  PROC Part73()
    MoveL Offs(pOrigin,152.4,74.3,0.0),vDraw,z1,tPen\WObj:=wPaper;
    MoveL Offs(pOrigin,152.2,74.1,0.0),vDraw,z1,tPen\WObj:=wPaper;
    MoveL Offs(pOrigin,152.2,73.8,0.0),vDraw,z1,tPen\WObj:=wPaper;
    MoveL Offs(pOrigin,152.0,73.6,0.0),vDraw,z1,tPen\WObj:=wPaper;
    MoveL Offs(pOrigin,152.0,73.0,0.0),vDraw,z1,tPen\WObj:=wPaper;
    MoveL Offs(pOrigin,151.8,72.8,0.0),vDraw,z1,tPen\WObj:=wPaper;
    MoveL Offs(pOrigin,151.8,72.4,0.0),vDraw,z1,tPen\WObj:=wPaper;
    MoveL Offs(pOrigin,151.6,72.2,0.0),vDraw,z1,tPen\WObj:=wPaper;
    MoveL Offs(pOrigin,151.6,71.9,0.0),vDraw,z1,tPen\WObj:=wPaper;
    MoveL Offs(pOrigin,151.4,71.7,0.0),vDraw,z1,tPen\WObj:=wPaper;
    MoveL Offs(pOrigin,151.4,71.3,0.0),vDraw,z1,tPen\WObj:=wPaper;
    MoveL Offs(pOrigin,151.3,71.1,0.0),vDraw,z1,tPen\WObj:=wPaper;
    MoveL Offs(pOrigin,151.3,70.7,0.0),vDraw,z1,tPen\WObj:=wPaper;
    MoveL Offs(pOrigin,151.1,70.5,0.0),vDraw,z1,tPen\WObj:=wPaper;
    MoveL Offs(pOrigin,151.1,70.0,0.0),vDraw,z1,tPen\WObj:=wPaper;
    MoveL Offs(pOrigin,150.9,69.8,0.0),vDraw,z1,tPen\WObj:=wPaper;
    MoveL Offs(pOrigin,150.9,69.4,0.0),vDraw,z1,tPen\WObj:=wPaper;
    MoveL Offs(pOrigin,150.7,69.2,0.0),vDraw,z1,tPen\WObj:=wPaper;
    MoveL Offs(pOrigin,150.7,68.8,0.0),vDraw,z1,tPen\WObj:=wPaper;
    MoveL Offs(pOrigin,150.5,68.7,0.0),vDraw,z1,tPen\WObj:=wPaper;
    MoveL Offs(pOrigin,150.5,68.3,0.0),vDraw,z1,tPen\WObj:=wPaper;
    MoveL Offs(pOrigin,150.3,68.1,0.0),vDraw,z1,tPen\WObj:=wPaper;
    MoveL Offs(pOrigin,150.3,67.7,0.0),vDraw,z1,tPen\WObj:=wPaper;
    MoveL Offs(pOrigin,150.1,67.5,0.0),vDraw,z1,tPen\WObj:=wPaper;
    MoveL Offs(pOrigin,150.1,67.0,0.0),vDraw,z1,tPen\WObj:=wPaper;
    MoveL Offs(pOrigin,149.9,66.8,0.0),vDraw,z1,tPen\WObj:=wPaper;
    MoveL Offs(pOrigin,149.9,66.4,0.0),vDraw,z1,tPen\WObj:=wPaper;
    MoveL Offs(pOrigin,149.7,66.2,0.0),vDraw,z1,tPen\WObj:=wPaper;
    MoveL Offs(pOrigin,149.7,65.8,0.0),vDraw,z1,tPen\WObj:=wPaper;
    MoveL Offs(pOrigin,149.6,65.6,0.0),vDraw,z1,tPen\WObj:=wPaper;
    MoveL Offs(pOrigin,149.6,65.3,0.0),vDraw,z1,tPen\WObj:=wPaper;
    MoveL Offs(pOrigin,149.4,65.1,0.0),vDraw,z1,tPen\WObj:=wPaper;
    MoveL Offs(pOrigin,149.4,64.7,0.0),vDraw,z1,tPen\WObj:=wPaper;
    MoveL Offs(pOrigin,149.2,64.5,0.0),vDraw,z1,tPen\WObj:=wPaper;
    MoveL Offs(pOrigin,149.2,64.1,0.0),vDraw,z1,tPen\WObj:=wPaper;
    MoveL Offs(pOrigin,149.0,63.9,0.0),vDraw,z1,tPen\WObj:=wPaper;
    MoveL Offs(pOrigin,149.0,63.6,0.0),vDraw,z1,tPen\WObj:=wPaper;
    MoveL Offs(pOrigin,148.8,63.4,0.0),vDraw,z1,tPen\WObj:=wPaper;
    MoveL Offs(pOrigin,148.8,63.0,0.0),vDraw,z1,tPen\WObj:=wPaper;
    MoveL Offs(pOrigin,148.6,62.8,0.0),vDraw,z1,tPen\WObj:=wPaper;
    MoveL Offs(pOrigin,148.6,62.4,0.0),vDraw,z1,tPen\WObj:=wPaper;
    MoveL Offs(pOrigin,148.4,62.2,0.0),vDraw,z1,tPen\WObj:=wPaper;
    MoveL Offs(pOrigin,148.4,61.7,0.0),vDraw,z1,tPen\WObj:=wPaper;
    MoveL Offs(pOrigin,148.2,61.5,0.0),vDraw,z1,tPen\WObj:=wPaper;
    MoveL Offs(pOrigin,148.2,61.1,0.0),vDraw,z1,tPen\WObj:=wPaper;
    MoveL Offs(pOrigin,148.0,60.9,0.0),vDraw,z1,tPen\WObj:=wPaper;
    MoveL Offs(pOrigin,148.0,60.5,0.0),vDraw,z1,tPen\WObj:=wPaper;
    MoveL Offs(pOrigin,147.9,60.3,0.0),vDraw,z1,tPen\WObj:=wPaper;
    MoveL Offs(pOrigin,147.9,59.8,0.0),vDraw,z1,tPen\WObj:=wPaper;
    MoveL Offs(pOrigin,147.5,59.2,0.0),vDraw,z1,tPen\WObj:=wPaper;
    MoveL Offs(pOrigin,147.5,58.6,0.0),vDraw,z1,tPen\WObj:=wPaper;
    MoveL Offs(pOrigin,147.3,58.5,0.0),vDraw,z1,tPen\WObj:=wPaper;
    MoveL Offs(pOrigin,147.3,58.1,0.0),vDraw,z1,tPen\WObj:=wPaper;
    MoveL Offs(pOrigin,147.1,57.9,0.0),vDraw,z1,tPen\WObj:=wPaper;
    MoveL Offs(pOrigin,147.1,57.5,0.0),vDraw,z1,tPen\WObj:=wPaper;
    MoveL Offs(pOrigin,146.9,57.3,0.0),vDraw,z1,tPen\WObj:=wPaper;
    MoveL Offs(pOrigin,146.9,56.9,0.0),vDraw,z1,tPen\WObj:=wPaper;
    MoveL Offs(pOrigin,146.7,56.8,0.0),vDraw,z1,tPen\WObj:=wPaper;
    MoveL Offs(pOrigin,146.7,56.2,0.0),vDraw,z1,tPen\WObj:=wPaper;
    MoveL Offs(pOrigin,146.5,56.0,0.0),vDraw,z1,tPen\WObj:=wPaper;
    MoveL Offs(pOrigin,146.5,55.6,0.0),vDraw,z1,tPen\WObj:=wPaper;
    MoveL Offs(pOrigin,146.3,55.4,0.0),vDraw,z1,tPen\WObj:=wPaper;
    MoveL Offs(pOrigin,146.3,55.1,0.0),vDraw,z1,tPen\WObj:=wPaper;
    MoveL Offs(pOrigin,146.2,54.9,0.0),vDraw,z1,tPen\WObj:=wPaper;
    MoveL Offs(pOrigin,146.2,54.3,0.0),vDraw,z1,tPen\WObj:=wPaper;
    MoveL Offs(pOrigin,146.0,54.1,0.0),vDraw,z1,tPen\WObj:=wPaper;
    MoveL Offs(pOrigin,146.0,53.7,0.0),vDraw,z1,tPen\WObj:=wPaper;
    MoveL Offs(pOrigin,145.8,53.5,0.0),vDraw,z1,tPen\WObj:=wPaper;
    MoveL Offs(pOrigin,145.8,53.0,0.0),vDraw,z1,tPen\WObj:=wPaper;
    MoveL Offs(pOrigin,145.6,52.8,0.0),vDraw,z1,tPen\WObj:=wPaper;
    MoveL Offs(pOrigin,145.6,52.2,0.0),vDraw,z1,tPen\WObj:=wPaper;
    MoveL Offs(pOrigin,145.4,52.0,0.0),vDraw,z1,tPen\WObj:=wPaper;
    MoveL Offs(pOrigin,145.4,51.5,0.0),vDraw,z1,tPen\WObj:=wPaper;
    MoveL Offs(pOrigin,145.2,51.3,0.0),vDraw,z1,tPen\WObj:=wPaper;
    MoveL Offs(pOrigin,145.2,50.9,0.0),vDraw,z1,tPen\WObj:=wPaper;
    MoveL Offs(pOrigin,145.0,50.7,0.0),vDraw,z1,tPen\WObj:=wPaper;
    MoveL Offs(pOrigin,145.0,50.1,0.0),vDraw,z1,tPen\WObj:=wPaper;
    MoveL Offs(pOrigin,144.8,50.0,0.0),vDraw,z1,tPen\WObj:=wPaper;
    MoveL Offs(pOrigin,144.8,49.4,0.0),vDraw,z1,tPen\WObj:=wPaper;
    MoveL Offs(pOrigin,144.6,49.2,0.0),vDraw,z1,tPen\WObj:=wPaper;
    MoveL Offs(pOrigin,144.6,48.6,0.0),vDraw,z1,tPen\WObj:=wPaper;
    MoveL Offs(pOrigin,144.5,48.4,0.0),vDraw,z1,tPen\WObj:=wPaper;
    MoveL Offs(pOrigin,144.5,47.7,0.0),vDraw,z1,tPen\WObj:=wPaper;
    MoveL Offs(pOrigin,144.3,47.5,0.0),vDraw,z1,tPen\WObj:=wPaper;
    MoveL Offs(pOrigin,144.3,46.9,0.0),vDraw,z1,tPen\WObj:=wPaper;
    MoveL Offs(pOrigin,144.1,46.7,0.0),vDraw,z1,tPen\WObj:=wPaper;
    MoveL Offs(pOrigin,144.1,46.2,0.0),vDraw,z1,tPen\WObj:=wPaper;
    MoveL Offs(pOrigin,143.9,46.0,0.0),vDraw,z1,tPen\WObj:=wPaper;
    MoveL Offs(pOrigin,143.9,45.2,0.0),vDraw,z1,tPen\WObj:=wPaper;
    MoveL Offs(pOrigin,143.7,45.0,0.0),vDraw,z1,tPen\WObj:=wPaper;
    MoveL Offs(pOrigin,143.7,44.3,0.0),vDraw,z1,tPen\WObj:=wPaper;
    MoveL Offs(pOrigin,143.5,44.1,0.0),vDraw,z1,tPen\WObj:=wPaper;
    MoveL Offs(pOrigin,143.5,43.3,0.0),vDraw,z1,tPen\WObj:=wPaper;
    MoveL Offs(pOrigin,143.3,43.2,0.0),vDraw,z1,tPen\WObj:=wPaper;
    MoveL Offs(pOrigin,143.3,42.4,0.0),vDraw,z1,tPen\WObj:=wPaper;
    MoveL Offs(pOrigin,143.1,42.2,0.0),vDraw,z1,tPen\WObj:=wPaper;
    MoveL Offs(pOrigin,143.1,41.3,0.0),vDraw,z1,tPen\WObj:=wPaper;
    MoveL Offs(pOrigin,142.9,41.1,0.0),vDraw,z1,tPen\WObj:=wPaper;
    MoveL Offs(pOrigin,142.9,40.1,0.0),vDraw,z1,tPen\WObj:=wPaper;
    MoveL Offs(pOrigin,142.8,39.9,0.0),vDraw,z1,tPen\WObj:=wPaper;
    MoveL Offs(pOrigin,142.8,39.0,0.0),vDraw,z1,tPen\WObj:=wPaper;
    MoveL Offs(pOrigin,142.6,38.8,0.0),vDraw,z1,tPen\WObj:=wPaper;
    MoveL Offs(pOrigin,142.6,37.5,0.0),vDraw,z1,tPen\WObj:=wPaper;
    MoveL Offs(pOrigin,142.0,36.7,0.0),vDraw,z1,tPen\WObj:=wPaper;
    MoveL Offs(pOrigin,140.3,36.7,0.0),vDraw,z1,tPen\WObj:=wPaper;
    MoveL Offs(pOrigin,140.1,36.5,0.0),vDraw,z1,tPen\WObj:=wPaper;
    MoveL Offs(pOrigin,139.2,36.4,0.0),vDraw,z1,tPen\WObj:=wPaper;
    MoveL Offs(pOrigin,138.2,35.8,0.0),vDraw,fine,tPen\WObj:=wPaper;
    MoveL Offs(pOrigin,138.2,35.8,15.0),vApproach,z5,tPen\WObj:=wPaper;
    MoveL Offs(pOrigin,143.1,36.7,15.0),vTravel,z5,tPen\WObj:=wPaper;
    MoveL Offs(pOrigin,143.1,36.7,0.0),vApproach,fine,tPen\WObj:=wPaper;
    MoveL Offs(pOrigin,143.1,37.3,0.0),vDraw,z1,tPen\WObj:=wPaper;
    MoveL Offs(pOrigin,143.3,37.5,0.0),vDraw,z1,tPen\WObj:=wPaper;
    MoveL Offs(pOrigin,143.3,38.8,0.0),vDraw,z1,tPen\WObj:=wPaper;
    MoveL Offs(pOrigin,143.5,39.0,0.0),vDraw,z1,tPen\WObj:=wPaper;
    MoveL Offs(pOrigin,143.5,40.1,0.0),vDraw,z1,tPen\WObj:=wPaper;
    MoveL Offs(pOrigin,143.7,40.3,0.0),vDraw,z1,tPen\WObj:=wPaper;
    MoveL Offs(pOrigin,143.7,41.1,0.0),vDraw,z1,tPen\WObj:=wPaper;
    MoveL Offs(pOrigin,143.9,41.3,0.0),vDraw,z1,tPen\WObj:=wPaper;
    MoveL Offs(pOrigin,143.9,42.2,0.0),vDraw,z1,tPen\WObj:=wPaper;
  ENDPROC

  PROC Part74()
    MoveL Offs(pOrigin,144.1,42.4,0.0),vDraw,z1,tPen\WObj:=wPaper;
    MoveL Offs(pOrigin,144.1,43.2,0.0),vDraw,z1,tPen\WObj:=wPaper;
    MoveL Offs(pOrigin,144.3,43.3,0.0),vDraw,z1,tPen\WObj:=wPaper;
    MoveL Offs(pOrigin,144.3,44.1,0.0),vDraw,z1,tPen\WObj:=wPaper;
    MoveL Offs(pOrigin,144.5,44.3,0.0),vDraw,z1,tPen\WObj:=wPaper;
    MoveL Offs(pOrigin,144.5,45.0,0.0),vDraw,z1,tPen\WObj:=wPaper;
    MoveL Offs(pOrigin,144.6,45.2,0.0),vDraw,z1,tPen\WObj:=wPaper;
    MoveL Offs(pOrigin,144.6,45.8,0.0),vDraw,z1,tPen\WObj:=wPaper;
    MoveL Offs(pOrigin,144.8,46.0,0.0),vDraw,z1,tPen\WObj:=wPaper;
    MoveL Offs(pOrigin,144.8,46.6,0.0),vDraw,z1,tPen\WObj:=wPaper;
    MoveL Offs(pOrigin,145.0,46.7,0.0),vDraw,z1,tPen\WObj:=wPaper;
    MoveL Offs(pOrigin,145.0,47.5,0.0),vDraw,z1,tPen\WObj:=wPaper;
    MoveL Offs(pOrigin,145.2,47.7,0.0),vDraw,z1,tPen\WObj:=wPaper;
    MoveL Offs(pOrigin,145.2,48.3,0.0),vDraw,z1,tPen\WObj:=wPaper;
    MoveL Offs(pOrigin,145.4,48.4,0.0),vDraw,z1,tPen\WObj:=wPaper;
    MoveL Offs(pOrigin,145.4,49.0,0.0),vDraw,z1,tPen\WObj:=wPaper;
    MoveL Offs(pOrigin,145.8,49.6,0.0),vDraw,z1,tPen\WObj:=wPaper;
    MoveL Offs(pOrigin,146.0,49.4,0.0),vDraw,z1,tPen\WObj:=wPaper;
    MoveL Offs(pOrigin,146.0,47.9,0.0),vDraw,z1,tPen\WObj:=wPaper;
    MoveL Offs(pOrigin,145.8,47.7,0.0),vDraw,z1,tPen\WObj:=wPaper;
    MoveL Offs(pOrigin,145.8,42.8,0.0),vDraw,z1,tPen\WObj:=wPaper;
    MoveL Offs(pOrigin,146.0,42.6,0.0),vDraw,z1,tPen\WObj:=wPaper;
    MoveL Offs(pOrigin,146.0,40.5,0.0),vDraw,z1,tPen\WObj:=wPaper;
    MoveL Offs(pOrigin,146.2,40.3,0.0),vDraw,z1,tPen\WObj:=wPaper;
    MoveL Offs(pOrigin,146.2,39.2,0.0),vDraw,z1,tPen\WObj:=wPaper;
    MoveL Offs(pOrigin,146.3,39.0,0.0),vDraw,z1,tPen\WObj:=wPaper;
    MoveL Offs(pOrigin,146.3,38.2,0.0),vDraw,z1,tPen\WObj:=wPaper;
    MoveL Offs(pOrigin,146.5,38.1,0.0),vDraw,z1,tPen\WObj:=wPaper;
    MoveL Offs(pOrigin,146.5,37.5,0.0),vDraw,z1,tPen\WObj:=wPaper;
    MoveL Offs(pOrigin,146.7,37.3,0.0),vDraw,z1,tPen\WObj:=wPaper;
    MoveL Offs(pOrigin,146.7,36.7,0.0),vDraw,z1,tPen\WObj:=wPaper;
    MoveL Offs(pOrigin,146.7,38.1,0.0),vDraw,z1,tPen\WObj:=wPaper;
    MoveL Offs(pOrigin,146.5,38.2,0.0),vDraw,z1,tPen\WObj:=wPaper;
    MoveL Offs(pOrigin,146.5,39.4,0.0),vDraw,z1,tPen\WObj:=wPaper;
    MoveL Offs(pOrigin,146.3,39.6,0.0),vDraw,z1,tPen\WObj:=wPaper;
    MoveL Offs(pOrigin,146.3,41.1,0.0),vDraw,z1,tPen\WObj:=wPaper;
    MoveL Offs(pOrigin,146.2,41.3,0.0),vDraw,z1,tPen\WObj:=wPaper;
    MoveL Offs(pOrigin,146.2,50.9,0.0),vDraw,z1,tPen\WObj:=wPaper;
    MoveL Offs(pOrigin,146.3,51.1,0.0),vDraw,z1,tPen\WObj:=wPaper;
    MoveL Offs(pOrigin,146.3,52.2,0.0),vDraw,z1,tPen\WObj:=wPaper;
    MoveL Offs(pOrigin,146.5,52.4,0.0),vDraw,z1,tPen\WObj:=wPaper;
    MoveL Offs(pOrigin,146.5,53.4,0.0),vDraw,z1,tPen\WObj:=wPaper;
    MoveL Offs(pOrigin,146.7,53.5,0.0),vDraw,z1,tPen\WObj:=wPaper;
    MoveL Offs(pOrigin,146.7,54.1,0.0),vDraw,z1,tPen\WObj:=wPaper;
    MoveL Offs(pOrigin,146.9,54.3,0.0),vDraw,z1,tPen\WObj:=wPaper;
    MoveL Offs(pOrigin,146.9,54.7,0.0),vDraw,z1,tPen\WObj:=wPaper;
    MoveL Offs(pOrigin,147.3,55.1,0.0),vDraw,z1,tPen\WObj:=wPaper;
    MoveL Offs(pOrigin,147.9,55.1,0.0),vDraw,z1,tPen\WObj:=wPaper;
    MoveL Offs(pOrigin,148.0,55.2,0.0),vDraw,z1,tPen\WObj:=wPaper;
    MoveL Offs(pOrigin,148.8,55.2,0.0),vDraw,z1,tPen\WObj:=wPaper;
    MoveL Offs(pOrigin,149.0,55.4,0.0),vDraw,z1,tPen\WObj:=wPaper;
    MoveL Offs(pOrigin,149.7,55.4,0.0),vDraw,z1,tPen\WObj:=wPaper;
    MoveL Offs(pOrigin,149.9,55.6,0.0),vDraw,z1,tPen\WObj:=wPaper;
    MoveL Offs(pOrigin,150.5,55.6,0.0),vDraw,z1,tPen\WObj:=wPaper;
    MoveL Offs(pOrigin,150.7,55.8,0.0),vDraw,z1,tPen\WObj:=wPaper;
    MoveL Offs(pOrigin,151.4,55.8,0.0),vDraw,z1,tPen\WObj:=wPaper;
    MoveL Offs(pOrigin,151.6,56.0,0.0),vDraw,z1,tPen\WObj:=wPaper;
    MoveL Offs(pOrigin,152.2,56.0,0.0),vDraw,z1,tPen\WObj:=wPaper;
    MoveL Offs(pOrigin,152.4,56.2,0.0),vDraw,z1,tPen\WObj:=wPaper;
    MoveL Offs(pOrigin,153.0,56.2,0.0),vDraw,z1,tPen\WObj:=wPaper;
    MoveL Offs(pOrigin,153.1,56.4,0.0),vDraw,z1,tPen\WObj:=wPaper;
    MoveL Offs(pOrigin,153.7,56.4,0.0),vDraw,z1,tPen\WObj:=wPaper;
    MoveL Offs(pOrigin,153.9,56.6,0.0),vDraw,z1,tPen\WObj:=wPaper;
    MoveL Offs(pOrigin,154.5,56.6,0.0),vDraw,z1,tPen\WObj:=wPaper;
    MoveL Offs(pOrigin,154.7,56.8,0.0),vDraw,z1,tPen\WObj:=wPaper;
    MoveL Offs(pOrigin,155.4,56.8,0.0),vDraw,z1,tPen\WObj:=wPaper;
    MoveL Offs(pOrigin,155.6,56.9,0.0),vDraw,z1,tPen\WObj:=wPaper;
    MoveL Offs(pOrigin,156.0,56.9,0.0),vDraw,z1,tPen\WObj:=wPaper;
    MoveL Offs(pOrigin,156.2,57.1,0.0),vDraw,z1,tPen\WObj:=wPaper;
    MoveL Offs(pOrigin,156.9,57.1,0.0),vDraw,z1,tPen\WObj:=wPaper;
    MoveL Offs(pOrigin,157.1,57.3,0.0),vDraw,z1,tPen\WObj:=wPaper;
    MoveL Offs(pOrigin,157.5,57.3,0.0),vDraw,z1,tPen\WObj:=wPaper;
    MoveL Offs(pOrigin,157.7,57.5,0.0),vDraw,z1,tPen\WObj:=wPaper;
    MoveL Offs(pOrigin,158.2,57.5,0.0),vDraw,z1,tPen\WObj:=wPaper;
    MoveL Offs(pOrigin,158.4,57.7,0.0),vDraw,z1,tPen\WObj:=wPaper;
    MoveL Offs(pOrigin,159.0,57.7,0.0),vDraw,z1,tPen\WObj:=wPaper;
    MoveL Offs(pOrigin,159.2,57.9,0.0),vDraw,z1,tPen\WObj:=wPaper;
    MoveL Offs(pOrigin,159.8,57.9,0.0),vDraw,z1,tPen\WObj:=wPaper;
    MoveL Offs(pOrigin,159.9,58.1,0.0),vDraw,z1,tPen\WObj:=wPaper;
    MoveL Offs(pOrigin,160.5,58.1,0.0),vDraw,z1,tPen\WObj:=wPaper;
    MoveL Offs(pOrigin,160.7,58.3,0.0),vDraw,z1,tPen\WObj:=wPaper;
    MoveL Offs(pOrigin,161.3,58.3,0.0),vDraw,z1,tPen\WObj:=wPaper;
    MoveL Offs(pOrigin,161.5,58.5,0.0),vDraw,z1,tPen\WObj:=wPaper;
    MoveL Offs(pOrigin,161.8,58.5,0.0),vDraw,z1,tPen\WObj:=wPaper;
    MoveL Offs(pOrigin,162.0,58.6,0.0),vDraw,z1,tPen\WObj:=wPaper;
    MoveL Offs(pOrigin,162.6,58.6,0.0),vDraw,z1,tPen\WObj:=wPaper;
    MoveL Offs(pOrigin,162.8,58.8,0.0),vDraw,z1,tPen\WObj:=wPaper;
    MoveL Offs(pOrigin,163.3,58.8,0.0),vDraw,z1,tPen\WObj:=wPaper;
    MoveL Offs(pOrigin,163.5,59.0,0.0),vDraw,z1,tPen\WObj:=wPaper;
    MoveL Offs(pOrigin,164.1,59.0,0.0),vDraw,z1,tPen\WObj:=wPaper;
    MoveL Offs(pOrigin,164.3,59.2,0.0),vDraw,z1,tPen\WObj:=wPaper;
    MoveL Offs(pOrigin,164.7,59.2,0.0),vDraw,z1,tPen\WObj:=wPaper;
    MoveL Offs(pOrigin,164.9,59.4,0.0),vDraw,z1,tPen\WObj:=wPaper;
    MoveL Offs(pOrigin,165.2,59.4,0.0),vDraw,z1,tPen\WObj:=wPaper;
    MoveL Offs(pOrigin,165.4,59.6,0.0),vDraw,z1,tPen\WObj:=wPaper;
    MoveL Offs(pOrigin,166.0,59.6,0.0),vDraw,z1,tPen\WObj:=wPaper;
    MoveL Offs(pOrigin,166.2,59.8,0.0),vDraw,z1,tPen\WObj:=wPaper;
    MoveL Offs(pOrigin,166.6,59.8,0.0),vDraw,z1,tPen\WObj:=wPaper;
    MoveL Offs(pOrigin,166.7,60.0,0.0),vDraw,z1,tPen\WObj:=wPaper;
    MoveL Offs(pOrigin,167.3,60.0,0.0),vDraw,z1,tPen\WObj:=wPaper;
    MoveL Offs(pOrigin,167.5,60.2,0.0),vDraw,z1,tPen\WObj:=wPaper;
    MoveL Offs(pOrigin,168.1,60.2,0.0),vDraw,z1,tPen\WObj:=wPaper;
    MoveL Offs(pOrigin,168.3,60.3,0.0),vDraw,z1,tPen\WObj:=wPaper;
    MoveL Offs(pOrigin,168.6,60.3,0.0),vDraw,z1,tPen\WObj:=wPaper;
    MoveL Offs(pOrigin,168.8,60.5,0.0),vDraw,z1,tPen\WObj:=wPaper;
    MoveL Offs(pOrigin,169.2,60.5,0.0),vDraw,z1,tPen\WObj:=wPaper;
    MoveL Offs(pOrigin,169.4,60.7,0.0),vDraw,z1,tPen\WObj:=wPaper;
    MoveL Offs(pOrigin,169.8,60.7,0.0),vDraw,z1,tPen\WObj:=wPaper;
    MoveL Offs(pOrigin,170.0,60.9,0.0),vDraw,z1,tPen\WObj:=wPaper;
    MoveL Offs(pOrigin,170.5,60.9,0.0),vDraw,z1,tPen\WObj:=wPaper;
    MoveL Offs(pOrigin,171.1,61.3,0.0),vDraw,z1,tPen\WObj:=wPaper;
    MoveL Offs(pOrigin,172.0,61.5,0.0),vDraw,z1,tPen\WObj:=wPaper;
    MoveL Offs(pOrigin,172.2,61.7,0.0),vDraw,z1,tPen\WObj:=wPaper;
    MoveL Offs(pOrigin,172.4,61.7,0.0),vDraw,z1,tPen\WObj:=wPaper;
    MoveL Offs(pOrigin,172.8,62.2,0.0),vDraw,z1,tPen\WObj:=wPaper;
    MoveL Offs(pOrigin,172.8,66.8,0.0),vDraw,z1,tPen\WObj:=wPaper;
    MoveL Offs(pOrigin,172.6,67.0,0.0),vDraw,z1,tPen\WObj:=wPaper;
    MoveL Offs(pOrigin,172.6,67.5,0.0),vDraw,z1,tPen\WObj:=wPaper;
    MoveL Offs(pOrigin,172.4,67.7,0.0),vDraw,z1,tPen\WObj:=wPaper;
    MoveL Offs(pOrigin,171.8,67.7,0.0),vDraw,z1,tPen\WObj:=wPaper;
  ENDPROC

  PROC Part75()
    MoveL Offs(pOrigin,171.7,67.5,0.0),vDraw,z1,tPen\WObj:=wPaper;
    MoveL Offs(pOrigin,171.3,67.5,0.0),vDraw,z1,tPen\WObj:=wPaper;
    MoveL Offs(pOrigin,171.1,67.3,0.0),vDraw,z1,tPen\WObj:=wPaper;
    MoveL Offs(pOrigin,170.7,67.3,0.0),vDraw,z1,tPen\WObj:=wPaper;
    MoveL Offs(pOrigin,170.5,67.1,0.0),vDraw,z1,tPen\WObj:=wPaper;
    MoveL Offs(pOrigin,170.0,67.1,0.0),vDraw,z1,tPen\WObj:=wPaper;
    MoveL Offs(pOrigin,169.8,67.0,0.0),vDraw,z1,tPen\WObj:=wPaper;
    MoveL Offs(pOrigin,169.4,67.0,0.0),vDraw,z1,tPen\WObj:=wPaper;
    MoveL Offs(pOrigin,169.2,66.8,0.0),vDraw,z1,tPen\WObj:=wPaper;
    MoveL Offs(pOrigin,168.8,66.8,0.0),vDraw,z1,tPen\WObj:=wPaper;
    MoveL Offs(pOrigin,168.6,66.6,0.0),vDraw,z1,tPen\WObj:=wPaper;
    MoveL Offs(pOrigin,168.1,66.6,0.0),vDraw,z1,tPen\WObj:=wPaper;
    MoveL Offs(pOrigin,167.9,66.4,0.0),vDraw,z1,tPen\WObj:=wPaper;
    MoveL Offs(pOrigin,167.7,66.4,0.0),vDraw,z1,tPen\WObj:=wPaper;
    MoveL Offs(pOrigin,167.5,66.6,0.0),vDraw,z1,tPen\WObj:=wPaper;
    MoveL Offs(pOrigin,168.8,67.9,0.0),vDraw,z1,tPen\WObj:=wPaper;
    MoveL Offs(pOrigin,169.0,67.9,0.0),vDraw,z1,tPen\WObj:=wPaper;
    MoveL Offs(pOrigin,169.8,68.7,0.0),vDraw,z1,tPen\WObj:=wPaper;
    MoveL Offs(pOrigin,170.0,68.7,0.0),vDraw,z1,tPen\WObj:=wPaper;
    MoveL Offs(pOrigin,170.7,69.4,0.0),vDraw,z1,tPen\WObj:=wPaper;
    MoveL Offs(pOrigin,170.9,69.4,0.0),vDraw,z1,tPen\WObj:=wPaper;
    MoveL Offs(pOrigin,171.5,70.0,0.0),vDraw,z1,tPen\WObj:=wPaper;
    MoveL Offs(pOrigin,171.7,70.0,0.0),vDraw,z1,tPen\WObj:=wPaper;
    MoveL Offs(pOrigin,172.4,70.7,0.0),vDraw,z1,tPen\WObj:=wPaper;
    MoveL Offs(pOrigin,172.6,70.7,0.0),vDraw,z1,tPen\WObj:=wPaper;
    MoveL Offs(pOrigin,173.0,71.1,0.0),vDraw,z1,tPen\WObj:=wPaper;
    MoveL Offs(pOrigin,172.8,70.9,0.0),vDraw,z1,tPen\WObj:=wPaper;
    MoveL Offs(pOrigin,171.8,70.5,0.0),vDraw,z1,tPen\WObj:=wPaper;
    MoveL Offs(pOrigin,171.5,70.2,0.0),vDraw,z1,tPen\WObj:=wPaper;
    MoveL Offs(pOrigin,171.3,70.2,0.0),vDraw,z1,tPen\WObj:=wPaper;
    MoveL Offs(pOrigin,170.9,69.8,0.0),vDraw,z1,tPen\WObj:=wPaper;
    MoveL Offs(pOrigin,170.7,69.8,0.0),vDraw,z1,tPen\WObj:=wPaper;
    MoveL Offs(pOrigin,170.3,69.4,0.0),vDraw,z1,tPen\WObj:=wPaper;
    MoveL Offs(pOrigin,170.1,69.4,0.0),vDraw,z1,tPen\WObj:=wPaper;
    MoveL Offs(pOrigin,168.3,67.7,0.0),vDraw,z1,tPen\WObj:=wPaper;
    MoveL Offs(pOrigin,168.1,67.7,0.0),vDraw,z1,tPen\WObj:=wPaper;
    MoveL Offs(pOrigin,166.4,66.0,0.0),vDraw,z1,tPen\WObj:=wPaper;
    MoveL Offs(pOrigin,166.2,66.0,0.0),vDraw,z1,tPen\WObj:=wPaper;
    MoveL Offs(pOrigin,166.0,65.8,0.0),vDraw,z1,tPen\WObj:=wPaper;
    MoveL Offs(pOrigin,165.4,65.8,0.0),vDraw,z1,tPen\WObj:=wPaper;
    MoveL Offs(pOrigin,165.2,65.6,0.0),vDraw,z1,tPen\WObj:=wPaper;
    MoveL Offs(pOrigin,164.9,65.6,0.0),vDraw,z1,tPen\WObj:=wPaper;
    MoveL Offs(pOrigin,164.7,65.4,0.0),vDraw,z1,tPen\WObj:=wPaper;
    MoveL Offs(pOrigin,164.1,65.4,0.0),vDraw,z1,tPen\WObj:=wPaper;
    MoveL Offs(pOrigin,163.9,65.3,0.0),vDraw,z1,tPen\WObj:=wPaper;
    MoveL Offs(pOrigin,163.5,65.3,0.0),vDraw,z1,tPen\WObj:=wPaper;
    MoveL Offs(pOrigin,163.3,65.1,0.0),vDraw,z1,tPen\WObj:=wPaper;
    MoveL Offs(pOrigin,162.8,65.1,0.0),vDraw,z1,tPen\WObj:=wPaper;
    MoveL Offs(pOrigin,162.6,64.9,0.0),vDraw,z1,tPen\WObj:=wPaper;
    MoveL Offs(pOrigin,162.0,64.9,0.0),vDraw,z1,tPen\WObj:=wPaper;
    MoveL Offs(pOrigin,161.8,64.7,0.0),vDraw,z1,tPen\WObj:=wPaper;
    MoveL Offs(pOrigin,161.5,64.7,0.0),vDraw,z1,tPen\WObj:=wPaper;
    MoveL Offs(pOrigin,161.3,64.5,0.0),vDraw,z1,tPen\WObj:=wPaper;
    MoveL Offs(pOrigin,160.9,64.5,0.0),vDraw,z1,tPen\WObj:=wPaper;
    MoveL Offs(pOrigin,160.7,64.3,0.0),vDraw,z1,tPen\WObj:=wPaper;
    MoveL Offs(pOrigin,160.1,64.3,0.0),vDraw,z1,tPen\WObj:=wPaper;
    MoveL Offs(pOrigin,159.9,64.1,0.0),vDraw,z1,tPen\WObj:=wPaper;
    MoveL Offs(pOrigin,159.4,64.1,0.0),vDraw,z1,tPen\WObj:=wPaper;
    MoveL Offs(pOrigin,159.2,63.9,0.0),vDraw,z1,tPen\WObj:=wPaper;
    MoveL Offs(pOrigin,158.8,63.9,0.0),vDraw,z1,tPen\WObj:=wPaper;
    MoveL Offs(pOrigin,158.6,63.7,0.0),vDraw,z1,tPen\WObj:=wPaper;
    MoveL Offs(pOrigin,158.1,63.7,0.0),vDraw,z1,tPen\WObj:=wPaper;
    MoveL Offs(pOrigin,157.9,63.6,0.0),vDraw,z1,tPen\WObj:=wPaper;
    MoveL Offs(pOrigin,157.3,63.6,0.0),vDraw,z1,tPen\WObj:=wPaper;
    MoveL Offs(pOrigin,157.1,63.4,0.0),vDraw,z1,tPen\WObj:=wPaper;
    MoveL Offs(pOrigin,156.7,63.4,0.0),vDraw,z1,tPen\WObj:=wPaper;
    MoveL Offs(pOrigin,156.5,63.2,0.0),vDraw,z1,tPen\WObj:=wPaper;
    MoveL Offs(pOrigin,156.2,63.2,0.0),vDraw,z1,tPen\WObj:=wPaper;
    MoveL Offs(pOrigin,156.0,63.0,0.0),vDraw,z1,tPen\WObj:=wPaper;
    MoveL Offs(pOrigin,155.4,63.0,0.0),vDraw,z1,tPen\WObj:=wPaper;
    MoveL Offs(pOrigin,155.2,62.8,0.0),vDraw,z1,tPen\WObj:=wPaper;
    MoveL Offs(pOrigin,154.7,62.8,0.0),vDraw,z1,tPen\WObj:=wPaper;
    MoveL Offs(pOrigin,154.5,62.6,0.0),vDraw,z1,tPen\WObj:=wPaper;
    MoveL Offs(pOrigin,154.1,62.6,0.0),vDraw,z1,tPen\WObj:=wPaper;
    MoveL Offs(pOrigin,153.9,62.4,0.0),vDraw,z1,tPen\WObj:=wPaper;
    MoveL Offs(pOrigin,153.3,62.4,0.0),vDraw,z1,tPen\WObj:=wPaper;
    MoveL Offs(pOrigin,153.1,62.2,0.0),vDraw,z1,tPen\WObj:=wPaper;
    MoveL Offs(pOrigin,152.8,62.2,0.0),vDraw,z1,tPen\WObj:=wPaper;
    MoveL Offs(pOrigin,152.6,62.0,0.0),vDraw,z1,tPen\WObj:=wPaper;
    MoveL Offs(pOrigin,152.0,62.0,0.0),vDraw,z1,tPen\WObj:=wPaper;
    MoveL Offs(pOrigin,151.8,61.9,0.0),vDraw,z1,tPen\WObj:=wPaper;
    MoveL Offs(pOrigin,151.4,61.9,0.0),vDraw,z1,tPen\WObj:=wPaper;
    MoveL Offs(pOrigin,151.3,61.7,0.0),vDraw,z1,tPen\WObj:=wPaper;
    MoveL Offs(pOrigin,150.7,61.7,0.0),vDraw,z1,tPen\WObj:=wPaper;
    MoveL Offs(pOrigin,150.5,61.5,0.0),vDraw,z1,tPen\WObj:=wPaper;
    MoveL Offs(pOrigin,149.9,61.5,0.0),vDraw,z1,tPen\WObj:=wPaper;
    MoveL Offs(pOrigin,149.7,61.3,0.0),vDraw,z1,tPen\WObj:=wPaper;
    MoveL Offs(pOrigin,149.4,61.3,0.0),vDraw,z1,tPen\WObj:=wPaper;
    MoveL Offs(pOrigin,149.2,61.5,0.0),vDraw,z1,tPen\WObj:=wPaper;
    MoveL Offs(pOrigin,149.2,62.0,0.0),vDraw,z1,tPen\WObj:=wPaper;
    MoveL Offs(pOrigin,149.4,62.2,0.0),vDraw,z1,tPen\WObj:=wPaper;
    MoveL Offs(pOrigin,149.4,62.6,0.0),vDraw,z1,tPen\WObj:=wPaper;
    MoveL Offs(pOrigin,149.6,62.8,0.0),vDraw,z1,tPen\WObj:=wPaper;
    MoveL Offs(pOrigin,149.6,63.2,0.0),vDraw,z1,tPen\WObj:=wPaper;
    MoveL Offs(pOrigin,149.7,63.4,0.0),vDraw,z1,tPen\WObj:=wPaper;
    MoveL Offs(pOrigin,149.7,63.7,0.0),vDraw,z1,tPen\WObj:=wPaper;
    MoveL Offs(pOrigin,149.9,63.9,0.0),vDraw,z1,tPen\WObj:=wPaper;
    MoveL Offs(pOrigin,149.9,64.3,0.0),vDraw,z1,tPen\WObj:=wPaper;
    MoveL Offs(pOrigin,150.1,64.5,0.0),vDraw,z1,tPen\WObj:=wPaper;
    MoveL Offs(pOrigin,150.1,64.9,0.0),vDraw,z1,tPen\WObj:=wPaper;
    MoveL Offs(pOrigin,150.3,65.1,0.0),vDraw,z1,tPen\WObj:=wPaper;
    MoveL Offs(pOrigin,150.3,65.6,0.0),vDraw,z1,tPen\WObj:=wPaper;
    MoveL Offs(pOrigin,150.5,65.8,0.0),vDraw,z1,tPen\WObj:=wPaper;
    MoveL Offs(pOrigin,150.5,66.2,0.0),vDraw,z1,tPen\WObj:=wPaper;
    MoveL Offs(pOrigin,150.7,66.4,0.0),vDraw,z1,tPen\WObj:=wPaper;
    MoveL Offs(pOrigin,150.7,66.8,0.0),vDraw,z1,tPen\WObj:=wPaper;
    MoveL Offs(pOrigin,150.9,67.0,0.0),vDraw,z1,tPen\WObj:=wPaper;
    MoveL Offs(pOrigin,150.9,67.3,0.0),vDraw,z1,tPen\WObj:=wPaper;
    MoveL Offs(pOrigin,151.1,67.5,0.0),vDraw,z1,tPen\WObj:=wPaper;
    MoveL Offs(pOrigin,151.1,67.9,0.0),vDraw,z1,tPen\WObj:=wPaper;
    MoveL Offs(pOrigin,151.3,68.1,0.0),vDraw,z1,tPen\WObj:=wPaper;
    MoveL Offs(pOrigin,151.3,68.7,0.0),vDraw,z1,tPen\WObj:=wPaper;
    MoveL Offs(pOrigin,151.4,68.8,0.0),vDraw,z1,tPen\WObj:=wPaper;
    MoveL Offs(pOrigin,151.4,69.2,0.0),vDraw,z1,tPen\WObj:=wPaper;
    MoveL Offs(pOrigin,151.6,69.4,0.0),vDraw,z1,tPen\WObj:=wPaper;
    MoveL Offs(pOrigin,151.6,69.8,0.0),vDraw,z1,tPen\WObj:=wPaper;
    MoveL Offs(pOrigin,151.8,70.0,0.0),vDraw,z1,tPen\WObj:=wPaper;
    MoveL Offs(pOrigin,151.8,70.4,0.0),vDraw,z1,tPen\WObj:=wPaper;
    MoveL Offs(pOrigin,152.0,70.5,0.0),vDraw,z1,tPen\WObj:=wPaper;
    MoveL Offs(pOrigin,152.0,70.9,0.0),vDraw,z1,tPen\WObj:=wPaper;
  ENDPROC

  PROC Part76()
    MoveL Offs(pOrigin,152.2,71.1,0.0),vDraw,z1,tPen\WObj:=wPaper;
    MoveL Offs(pOrigin,152.2,71.7,0.0),vDraw,z1,tPen\WObj:=wPaper;
    MoveL Offs(pOrigin,152.4,71.9,0.0),vDraw,z1,tPen\WObj:=wPaper;
    MoveL Offs(pOrigin,152.4,72.2,0.0),vDraw,z1,tPen\WObj:=wPaper;
    MoveL Offs(pOrigin,152.6,72.4,0.0),vDraw,z1,tPen\WObj:=wPaper;
    MoveL Offs(pOrigin,152.6,72.8,0.0),vDraw,z1,tPen\WObj:=wPaper;
    MoveL Offs(pOrigin,152.8,73.0,0.0),vDraw,z1,tPen\WObj:=wPaper;
    MoveL Offs(pOrigin,152.8,73.4,0.0),vDraw,z1,tPen\WObj:=wPaper;
    MoveL Offs(pOrigin,153.0,73.6,0.0),vDraw,z1,tPen\WObj:=wPaper;
    MoveL Offs(pOrigin,153.0,74.1,0.0),vDraw,z1,tPen\WObj:=wPaper;
    MoveL Offs(pOrigin,153.1,74.3,0.0),vDraw,z1,tPen\WObj:=wPaper;
    MoveL Offs(pOrigin,153.1,74.7,0.0),vDraw,z1,tPen\WObj:=wPaper;
    MoveL Offs(pOrigin,153.3,74.9,0.0),vDraw,z1,tPen\WObj:=wPaper;
    MoveL Offs(pOrigin,153.3,75.3,0.0),vDraw,z1,tPen\WObj:=wPaper;
    MoveL Offs(pOrigin,153.5,75.5,0.0),vDraw,z1,tPen\WObj:=wPaper;
    MoveL Offs(pOrigin,153.5,75.8,0.0),vDraw,z1,tPen\WObj:=wPaper;
    MoveL Offs(pOrigin,153.7,76.0,0.0),vDraw,z1,tPen\WObj:=wPaper;
    MoveL Offs(pOrigin,153.7,76.4,0.0),vDraw,z1,tPen\WObj:=wPaper;
    MoveL Offs(pOrigin,153.9,76.6,0.0),vDraw,z1,tPen\WObj:=wPaper;
    MoveL Offs(pOrigin,153.9,77.2,0.0),vDraw,z1,tPen\WObj:=wPaper;
    MoveL Offs(pOrigin,154.1,77.3,0.0),vDraw,z1,tPen\WObj:=wPaper;
    MoveL Offs(pOrigin,154.1,77.7,0.0),vDraw,z1,tPen\WObj:=wPaper;
    MoveL Offs(pOrigin,154.3,77.9,0.0),vDraw,z1,tPen\WObj:=wPaper;
    MoveL Offs(pOrigin,154.3,78.3,0.0),vDraw,z1,tPen\WObj:=wPaper;
    MoveL Offs(pOrigin,154.5,78.5,0.0),vDraw,z1,tPen\WObj:=wPaper;
    MoveL Offs(pOrigin,154.5,78.9,0.0),vDraw,z1,tPen\WObj:=wPaper;
    MoveL Offs(pOrigin,154.7,79.0,0.0),vDraw,z1,tPen\WObj:=wPaper;
    MoveL Offs(pOrigin,154.7,79.4,0.0),vDraw,z1,tPen\WObj:=wPaper;
    MoveL Offs(pOrigin,154.8,79.6,0.0),vDraw,z1,tPen\WObj:=wPaper;
    MoveL Offs(pOrigin,154.8,80.2,0.0),vDraw,z1,tPen\WObj:=wPaper;
    MoveL Offs(pOrigin,155.0,80.4,0.0),vDraw,z1,tPen\WObj:=wPaper;
    MoveL Offs(pOrigin,155.0,80.7,0.0),vDraw,z1,tPen\WObj:=wPaper;
    MoveL Offs(pOrigin,155.2,80.9,0.0),vDraw,z1,tPen\WObj:=wPaper;
    MoveL Offs(pOrigin,155.2,81.3,0.0),vDraw,z1,tPen\WObj:=wPaper;
    MoveL Offs(pOrigin,155.4,81.5,0.0),vDraw,z1,tPen\WObj:=wPaper;
    MoveL Offs(pOrigin,155.4,81.9,0.0),vDraw,z1,tPen\WObj:=wPaper;
    MoveL Offs(pOrigin,155.6,82.1,0.0),vDraw,z1,tPen\WObj:=wPaper;
    MoveL Offs(pOrigin,155.6,82.4,0.0),vDraw,z1,tPen\WObj:=wPaper;
    MoveL Offs(pOrigin,155.8,82.6,0.0),vDraw,z1,tPen\WObj:=wPaper;
    MoveL Offs(pOrigin,155.8,83.0,0.0),vDraw,z1,tPen\WObj:=wPaper;
    MoveL Offs(pOrigin,156.0,83.2,0.0),vDraw,z1,tPen\WObj:=wPaper;
    MoveL Offs(pOrigin,156.0,83.6,0.0),vDraw,z1,tPen\WObj:=wPaper;
    MoveL Offs(pOrigin,156.2,83.8,0.0),vDraw,z1,tPen\WObj:=wPaper;
    MoveL Offs(pOrigin,156.2,84.3,0.0),vDraw,z1,tPen\WObj:=wPaper;
    MoveL Offs(pOrigin,156.4,84.5,0.0),vDraw,z1,tPen\WObj:=wPaper;
    MoveL Offs(pOrigin,156.4,84.9,0.0),vDraw,z1,tPen\WObj:=wPaper;
    MoveL Offs(pOrigin,156.5,85.1,0.0),vDraw,z1,tPen\WObj:=wPaper;
    MoveL Offs(pOrigin,156.5,85.5,0.0),vDraw,z1,tPen\WObj:=wPaper;
    MoveL Offs(pOrigin,156.7,85.7,0.0),vDraw,z1,tPen\WObj:=wPaper;
    MoveL Offs(pOrigin,156.7,86.0,0.0),vDraw,z1,tPen\WObj:=wPaper;
    MoveL Offs(pOrigin,156.9,86.2,0.0),vDraw,z1,tPen\WObj:=wPaper;
    MoveL Offs(pOrigin,156.9,86.6,0.0),vDraw,z1,tPen\WObj:=wPaper;
    MoveL Offs(pOrigin,157.1,86.8,0.0),vDraw,z1,tPen\WObj:=wPaper;
    MoveL Offs(pOrigin,157.1,87.2,0.0),vDraw,z1,tPen\WObj:=wPaper;
    MoveL Offs(pOrigin,157.3,87.4,0.0),vDraw,z1,tPen\WObj:=wPaper;
    MoveL Offs(pOrigin,157.3,87.7,0.0),vDraw,z1,tPen\WObj:=wPaper;
    MoveL Offs(pOrigin,157.5,87.9,0.0),vDraw,z1,tPen\WObj:=wPaper;
    MoveL Offs(pOrigin,157.5,88.3,0.0),vDraw,z1,tPen\WObj:=wPaper;
    MoveL Offs(pOrigin,157.7,88.5,0.0),vDraw,z1,tPen\WObj:=wPaper;
    MoveL Offs(pOrigin,157.7,88.9,0.0),vDraw,z1,tPen\WObj:=wPaper;
    MoveL Offs(pOrigin,157.9,89.1,0.0),vDraw,z1,tPen\WObj:=wPaper;
    MoveL Offs(pOrigin,157.9,89.4,0.0),vDraw,z1,tPen\WObj:=wPaper;
    MoveL Offs(pOrigin,158.1,89.6,0.0),vDraw,z1,tPen\WObj:=wPaper;
    MoveL Offs(pOrigin,158.1,90.0,0.0),vDraw,z1,tPen\WObj:=wPaper;
    MoveL Offs(pOrigin,158.2,90.2,0.0),vDraw,z1,tPen\WObj:=wPaper;
    MoveL Offs(pOrigin,158.2,90.6,0.0),vDraw,z1,tPen\WObj:=wPaper;
    MoveL Offs(pOrigin,158.4,90.8,0.0),vDraw,z1,tPen\WObj:=wPaper;
    MoveL Offs(pOrigin,158.4,91.1,0.0),vDraw,z1,tPen\WObj:=wPaper;
    MoveL Offs(pOrigin,158.6,91.3,0.0),vDraw,z1,tPen\WObj:=wPaper;
    MoveL Offs(pOrigin,158.6,91.7,0.0),vDraw,z1,tPen\WObj:=wPaper;
    MoveL Offs(pOrigin,158.8,91.9,0.0),vDraw,z1,tPen\WObj:=wPaper;
    MoveL Offs(pOrigin,158.8,92.3,0.0),vDraw,z1,tPen\WObj:=wPaper;
    MoveL Offs(pOrigin,159.0,92.5,0.0),vDraw,z1,tPen\WObj:=wPaper;
    MoveL Offs(pOrigin,159.0,92.8,0.0),vDraw,z1,tPen\WObj:=wPaper;
    MoveL Offs(pOrigin,159.2,93.0,0.0),vDraw,z1,tPen\WObj:=wPaper;
    MoveL Offs(pOrigin,159.2,94.0,0.0),vDraw,z1,tPen\WObj:=wPaper;
    MoveL Offs(pOrigin,159.0,94.2,0.0),vDraw,z1,tPen\WObj:=wPaper;
    MoveL Offs(pOrigin,158.8,94.2,0.0),vDraw,z1,tPen\WObj:=wPaper;
    MoveL Offs(pOrigin,158.6,94.3,0.0),vDraw,z1,tPen\WObj:=wPaper;
    MoveL Offs(pOrigin,158.2,94.3,0.0),vDraw,z1,tPen\WObj:=wPaper;
    MoveL Offs(pOrigin,158.1,94.5,0.0),vDraw,z1,tPen\WObj:=wPaper;
    MoveL Offs(pOrigin,157.7,94.5,0.0),vDraw,z1,tPen\WObj:=wPaper;
    MoveL Offs(pOrigin,157.5,94.7,0.0),vDraw,z1,tPen\WObj:=wPaper;
    MoveL Offs(pOrigin,157.1,94.7,0.0),vDraw,z1,tPen\WObj:=wPaper;
    MoveL Offs(pOrigin,156.9,94.9,0.0),vDraw,z1,tPen\WObj:=wPaper;
    MoveL Offs(pOrigin,156.5,94.9,0.0),vDraw,z1,tPen\WObj:=wPaper;
    MoveL Offs(pOrigin,156.4,95.1,0.0),vDraw,z1,tPen\WObj:=wPaper;
    MoveL Offs(pOrigin,156.0,95.1,0.0),vDraw,z1,tPen\WObj:=wPaper;
    MoveL Offs(pOrigin,155.8,95.3,0.0),vDraw,z1,tPen\WObj:=wPaper;
    MoveL Offs(pOrigin,155.4,95.3,0.0),vDraw,z1,tPen\WObj:=wPaper;
    MoveL Offs(pOrigin,155.2,95.5,0.0),vDraw,z1,tPen\WObj:=wPaper;
    MoveL Offs(pOrigin,154.8,95.5,0.0),vDraw,z1,tPen\WObj:=wPaper;
    MoveL Offs(pOrigin,154.7,95.7,0.0),vDraw,z1,tPen\WObj:=wPaper;
    MoveL Offs(pOrigin,154.3,95.7,0.0),vDraw,z1,tPen\WObj:=wPaper;
    MoveL Offs(pOrigin,154.1,95.9,0.0),vDraw,z1,tPen\WObj:=wPaper;
    MoveL Offs(pOrigin,153.7,95.9,0.0),vDraw,z1,tPen\WObj:=wPaper;
    MoveL Offs(pOrigin,153.5,96.0,0.0),vDraw,z1,tPen\WObj:=wPaper;
    MoveL Offs(pOrigin,153.1,96.0,0.0),vDraw,z1,tPen\WObj:=wPaper;
    MoveL Offs(pOrigin,152.6,96.4,0.0),vDraw,z1,tPen\WObj:=wPaper;
    MoveL Offs(pOrigin,152.2,96.4,0.0),vDraw,z1,tPen\WObj:=wPaper;
    MoveL Offs(pOrigin,152.0,96.6,0.0),vDraw,z1,tPen\WObj:=wPaper;
    MoveL Offs(pOrigin,152.0,96.8,0.0),vDraw,z1,tPen\WObj:=wPaper;
    MoveL Offs(pOrigin,152.4,97.2,0.0),vDraw,z1,tPen\WObj:=wPaper;
    MoveL Offs(pOrigin,152.6,97.2,0.0),vDraw,z1,tPen\WObj:=wPaper;
    MoveL Offs(pOrigin,153.5,97.7,0.0),vDraw,z1,tPen\WObj:=wPaper;
    MoveL Offs(pOrigin,153.9,97.7,0.0),vDraw,z1,tPen\WObj:=wPaper;
    MoveL Offs(pOrigin,154.1,97.9,0.0),vDraw,z1,tPen\WObj:=wPaper;
    MoveL Offs(pOrigin,154.3,97.9,0.0),vDraw,z1,tPen\WObj:=wPaper;
    MoveL Offs(pOrigin,154.5,98.1,0.0),vDraw,z1,tPen\WObj:=wPaper;
    MoveL Offs(pOrigin,154.7,98.1,0.0),vDraw,z1,tPen\WObj:=wPaper;
    MoveL Offs(pOrigin,156.7,99.3,0.0),vDraw,z1,tPen\WObj:=wPaper;
    MoveL Offs(pOrigin,157.1,99.3,0.0),vDraw,z1,tPen\WObj:=wPaper;
    MoveL Offs(pOrigin,157.9,99.8,0.0),vDraw,z1,tPen\WObj:=wPaper;
    MoveL Offs(pOrigin,158.2,99.8,0.0),vDraw,z1,tPen\WObj:=wPaper;
    MoveL Offs(pOrigin,158.4,99.6,0.0),vDraw,z1,tPen\WObj:=wPaper;
    MoveL Offs(pOrigin,158.4,99.4,0.0),vDraw,z1,tPen\WObj:=wPaper;
    MoveL Offs(pOrigin,159.6,97.4,0.0),vDraw,z1,tPen\WObj:=wPaper;
    MoveL Offs(pOrigin,159.6,97.0,0.0),vDraw,z1,tPen\WObj:=wPaper;
    MoveL Offs(pOrigin,159.8,96.8,0.0),vDraw,z1,tPen\WObj:=wPaper;
    MoveL Offs(pOrigin,159.8,96.2,0.0),vDraw,z1,tPen\WObj:=wPaper;
  ENDPROC

  PROC Part77()
    MoveL Offs(pOrigin,159.9,96.0,0.0),vDraw,z1,tPen\WObj:=wPaper;
    MoveL Offs(pOrigin,159.9,95.3,0.0),vDraw,z1,tPen\WObj:=wPaper;
    MoveL Offs(pOrigin,160.1,95.1,0.0),vDraw,z1,tPen\WObj:=wPaper;
    MoveL Offs(pOrigin,160.1,92.3,0.0),vDraw,z1,tPen\WObj:=wPaper;
    MoveL Offs(pOrigin,159.9,92.1,0.0),vDraw,z1,tPen\WObj:=wPaper;
    MoveL Offs(pOrigin,159.9,91.1,0.0),vDraw,z1,tPen\WObj:=wPaper;
    MoveL Offs(pOrigin,159.8,90.9,0.0),vDraw,z1,tPen\WObj:=wPaper;
    MoveL Offs(pOrigin,159.8,90.0,0.0),vDraw,z1,tPen\WObj:=wPaper;
    MoveL Offs(pOrigin,159.8,90.2,0.0),vDraw,z1,tPen\WObj:=wPaper;
    MoveL Offs(pOrigin,159.9,90.4,0.0),vDraw,z1,tPen\WObj:=wPaper;
    MoveL Offs(pOrigin,159.9,90.9,0.0),vDraw,z1,tPen\WObj:=wPaper;
    MoveL Offs(pOrigin,160.1,91.1,0.0),vDraw,z1,tPen\WObj:=wPaper;
    MoveL Offs(pOrigin,160.1,91.5,0.0),vDraw,z1,tPen\WObj:=wPaper;
    MoveL Offs(pOrigin,160.3,91.7,0.0),vDraw,z1,tPen\WObj:=wPaper;
    MoveL Offs(pOrigin,160.3,93.0,0.0),vDraw,z1,tPen\WObj:=wPaper;
    MoveL Offs(pOrigin,160.5,93.2,0.0),vDraw,z1,tPen\WObj:=wPaper;
    MoveL Offs(pOrigin,160.5,94.7,0.0),vDraw,z1,tPen\WObj:=wPaper;
    MoveL Offs(pOrigin,160.3,94.9,0.0),vDraw,z1,tPen\WObj:=wPaper;
    MoveL Offs(pOrigin,160.3,95.9,0.0),vDraw,z1,tPen\WObj:=wPaper;
    MoveL Offs(pOrigin,160.1,96.0,0.0),vDraw,z1,tPen\WObj:=wPaper;
    MoveL Offs(pOrigin,160.1,96.6,0.0),vDraw,z1,tPen\WObj:=wPaper;
    MoveL Offs(pOrigin,159.9,96.8,0.0),vDraw,z1,tPen\WObj:=wPaper;
    MoveL Offs(pOrigin,159.9,97.2,0.0),vDraw,z1,tPen\WObj:=wPaper;
    MoveL Offs(pOrigin,159.6,97.7,0.0),vDraw,z1,tPen\WObj:=wPaper;
    MoveL Offs(pOrigin,159.6,98.1,0.0),vDraw,z1,tPen\WObj:=wPaper;
    MoveL Offs(pOrigin,159.0,98.9,0.0),vDraw,z1,tPen\WObj:=wPaper;
    MoveL Offs(pOrigin,159.0,99.1,0.0),vDraw,z1,tPen\WObj:=wPaper;
    MoveL Offs(pOrigin,158.4,99.6,0.0),vDraw,z1,tPen\WObj:=wPaper;
    MoveL Offs(pOrigin,158.4,99.8,0.0),vDraw,z1,tPen\WObj:=wPaper;
    MoveL Offs(pOrigin,158.1,100.2,0.0),vDraw,z1,tPen\WObj:=wPaper;
    MoveL Offs(pOrigin,158.1,100.4,0.0),vDraw,z1,tPen\WObj:=wPaper;
    MoveL Offs(pOrigin,157.3,101.1,0.0),vDraw,z1,tPen\WObj:=wPaper;
    MoveL Offs(pOrigin,157.1,101.1,0.0),vDraw,z1,tPen\WObj:=wPaper;
    MoveL Offs(pOrigin,156.7,101.5,0.0),vDraw,z1,tPen\WObj:=wPaper;
    MoveL Offs(pOrigin,156.7,101.7,0.0),vDraw,z1,tPen\WObj:=wPaper;
    MoveL Offs(pOrigin,155.2,103.4,0.0),vDraw,z1,tPen\WObj:=wPaper;
    MoveL Offs(pOrigin,155.2,103.6,0.0),vDraw,z1,tPen\WObj:=wPaper;
    MoveL Offs(pOrigin,154.7,104.2,0.0),vDraw,z1,tPen\WObj:=wPaper;
    MoveL Offs(pOrigin,154.7,104.4,0.0),vDraw,z1,tPen\WObj:=wPaper;
    MoveL Offs(pOrigin,154.8,104.5,0.0),vDraw,z1,tPen\WObj:=wPaper;
    MoveL Offs(pOrigin,155.4,104.5,0.0),vDraw,z1,tPen\WObj:=wPaper;
    MoveL Offs(pOrigin,155.6,104.4,0.0),vDraw,z1,tPen\WObj:=wPaper;
    MoveL Offs(pOrigin,156.4,104.4,0.0),vDraw,z1,tPen\WObj:=wPaper;
    MoveL Offs(pOrigin,156.5,104.2,0.0),vDraw,z1,tPen\WObj:=wPaper;
    MoveL Offs(pOrigin,157.1,104.2,0.0),vDraw,z1,tPen\WObj:=wPaper;
    MoveL Offs(pOrigin,157.3,104.0,0.0),vDraw,z1,tPen\WObj:=wPaper;
    MoveL Offs(pOrigin,157.9,104.0,0.0),vDraw,z1,tPen\WObj:=wPaper;
    MoveL Offs(pOrigin,158.1,103.8,0.0),vDraw,z1,tPen\WObj:=wPaper;
    MoveL Offs(pOrigin,158.6,103.8,0.0),vDraw,z1,tPen\WObj:=wPaper;
    MoveL Offs(pOrigin,158.8,103.6,0.0),vDraw,z1,tPen\WObj:=wPaper;
    MoveL Offs(pOrigin,159.4,103.6,0.0),vDraw,z1,tPen\WObj:=wPaper;
    MoveL Offs(pOrigin,159.6,103.4,0.0),vDraw,z1,tPen\WObj:=wPaper;
    MoveL Offs(pOrigin,159.9,103.4,0.0),vDraw,z1,tPen\WObj:=wPaper;
    MoveL Offs(pOrigin,160.1,103.2,0.0),vDraw,z1,tPen\WObj:=wPaper;
    MoveL Offs(pOrigin,160.7,103.2,0.0),vDraw,z1,tPen\WObj:=wPaper;
    MoveL Offs(pOrigin,160.9,103.0,0.0),vDraw,z1,tPen\WObj:=wPaper;
    MoveL Offs(pOrigin,161.3,103.0,0.0),vDraw,z1,tPen\WObj:=wPaper;
    MoveL Offs(pOrigin,161.5,102.8,0.0),vDraw,z1,tPen\WObj:=wPaper;
    MoveL Offs(pOrigin,161.8,102.8,0.0),vDraw,z1,tPen\WObj:=wPaper;
    MoveL Offs(pOrigin,162.0,102.7,0.0),vDraw,z1,tPen\WObj:=wPaper;
    MoveL Offs(pOrigin,162.4,102.7,0.0),vDraw,z1,tPen\WObj:=wPaper;
    MoveL Offs(pOrigin,162.6,102.5,0.0),vDraw,z1,tPen\WObj:=wPaper;
    MoveL Offs(pOrigin,163.0,102.5,0.0),vDraw,z1,tPen\WObj:=wPaper;
    MoveL Offs(pOrigin,163.2,102.3,0.0),vDraw,z1,tPen\WObj:=wPaper;
    MoveL Offs(pOrigin,163.5,102.3,0.0),vDraw,z1,tPen\WObj:=wPaper;
    MoveL Offs(pOrigin,163.7,102.1,0.0),vDraw,z1,tPen\WObj:=wPaper;
    MoveL Offs(pOrigin,164.1,102.1,0.0),vDraw,z1,tPen\WObj:=wPaper;
    MoveL Offs(pOrigin,164.3,101.9,0.0),vDraw,z1,tPen\WObj:=wPaper;
    MoveL Offs(pOrigin,164.7,101.9,0.0),vDraw,z1,tPen\WObj:=wPaper;
    MoveL Offs(pOrigin,164.9,101.7,0.0),vDraw,z1,tPen\WObj:=wPaper;
    MoveL Offs(pOrigin,165.2,101.7,0.0),vDraw,z1,tPen\WObj:=wPaper;
    MoveL Offs(pOrigin,165.4,101.5,0.0),vDraw,z1,tPen\WObj:=wPaper;
    MoveL Offs(pOrigin,166.0,101.5,0.0),vDraw,z1,tPen\WObj:=wPaper;
    MoveL Offs(pOrigin,165.8,101.5,0.0),vDraw,z1,tPen\WObj:=wPaper;
    MoveL Offs(pOrigin,165.2,101.9,0.0),vDraw,z1,tPen\WObj:=wPaper;
    MoveL Offs(pOrigin,164.3,102.1,0.0),vDraw,z1,tPen\WObj:=wPaper;
    MoveL Offs(pOrigin,163.3,102.7,0.0),vDraw,z1,tPen\WObj:=wPaper;
    MoveL Offs(pOrigin,162.4,102.8,0.0),vDraw,z1,tPen\WObj:=wPaper;
    MoveL Offs(pOrigin,161.8,103.2,0.0),vDraw,z1,tPen\WObj:=wPaper;
    MoveL Offs(pOrigin,161.5,103.2,0.0),vDraw,z1,tPen\WObj:=wPaper;
    MoveL Offs(pOrigin,161.3,103.4,0.0),vDraw,z1,tPen\WObj:=wPaper;
    MoveL Offs(pOrigin,160.9,103.4,0.0),vDraw,z1,tPen\WObj:=wPaper;
    MoveL Offs(pOrigin,160.7,103.6,0.0),vDraw,z1,tPen\WObj:=wPaper;
    MoveL Offs(pOrigin,160.3,103.6,0.0),vDraw,z1,tPen\WObj:=wPaper;
    MoveL Offs(pOrigin,160.1,103.8,0.0),vDraw,z1,tPen\WObj:=wPaper;
    MoveL Offs(pOrigin,159.8,103.8,0.0),vDraw,z1,tPen\WObj:=wPaper;
    MoveL Offs(pOrigin,159.6,104.0,0.0),vDraw,z1,tPen\WObj:=wPaper;
    MoveL Offs(pOrigin,159.2,104.0,0.0),vDraw,z1,tPen\WObj:=wPaper;
    MoveL Offs(pOrigin,159.0,104.2,0.0),vDraw,z1,tPen\WObj:=wPaper;
    MoveL Offs(pOrigin,158.6,104.2,0.0),vDraw,z1,tPen\WObj:=wPaper;
    MoveL Offs(pOrigin,158.4,104.4,0.0),vDraw,z1,tPen\WObj:=wPaper;
    MoveL Offs(pOrigin,157.9,104.4,0.0),vDraw,z1,tPen\WObj:=wPaper;
    MoveL Offs(pOrigin,157.7,104.5,0.0),vDraw,z1,tPen\WObj:=wPaper;
    MoveL Offs(pOrigin,157.1,104.5,0.0),vDraw,z1,tPen\WObj:=wPaper;
    MoveL Offs(pOrigin,156.9,104.7,0.0),vDraw,z1,tPen\WObj:=wPaper;
    MoveL Offs(pOrigin,156.2,104.7,0.0),vDraw,z1,tPen\WObj:=wPaper;
    MoveL Offs(pOrigin,156.0,104.9,0.0),vDraw,z1,tPen\WObj:=wPaper;
    MoveL Offs(pOrigin,155.0,104.9,0.0),vDraw,z1,tPen\WObj:=wPaper;
    MoveL Offs(pOrigin,154.8,105.1,0.0),vDraw,z1,tPen\WObj:=wPaper;
    MoveL Offs(pOrigin,154.1,105.1,0.0),vDraw,z1,tPen\WObj:=wPaper;
    MoveL Offs(pOrigin,153.1,106.1,0.0),vDraw,z1,tPen\WObj:=wPaper;
    MoveL Offs(pOrigin,153.1,106.2,0.0),vDraw,z1,tPen\WObj:=wPaper;
    MoveL Offs(pOrigin,152.2,107.2,0.0),vDraw,z1,tPen\WObj:=wPaper;
    MoveL Offs(pOrigin,152.2,107.4,0.0),vDraw,z1,tPen\WObj:=wPaper;
    MoveL Offs(pOrigin,151.6,107.9,0.0),vDraw,z1,tPen\WObj:=wPaper;
    MoveL Offs(pOrigin,151.6,108.1,0.0),vDraw,z1,tPen\WObj:=wPaper;
    MoveL Offs(pOrigin,151.8,108.3,0.0),vDraw,z1,tPen\WObj:=wPaper;
    MoveL Offs(pOrigin,152.0,108.3,0.0),vDraw,z1,tPen\WObj:=wPaper;
    MoveL Offs(pOrigin,152.2,108.1,0.0),vDraw,z1,tPen\WObj:=wPaper;
    MoveL Offs(pOrigin,152.8,108.1,0.0),vDraw,z1,tPen\WObj:=wPaper;
    MoveL Offs(pOrigin,153.0,107.9,0.0),vDraw,z1,tPen\WObj:=wPaper;
    MoveL Offs(pOrigin,153.5,107.9,0.0),vDraw,z1,tPen\WObj:=wPaper;
    MoveL Offs(pOrigin,153.7,107.8,0.0),vDraw,z1,tPen\WObj:=wPaper;
    MoveL Offs(pOrigin,154.3,107.8,0.0),vDraw,z1,tPen\WObj:=wPaper;
    MoveL Offs(pOrigin,154.5,107.6,0.0),vDraw,z1,tPen\WObj:=wPaper;
    MoveL Offs(pOrigin,154.8,107.6,0.0),vDraw,z1,tPen\WObj:=wPaper;
    MoveL Offs(pOrigin,155.0,107.4,0.0),vDraw,z1,tPen\WObj:=wPaper;
    MoveL Offs(pOrigin,155.4,107.4,0.0),vDraw,z1,tPen\WObj:=wPaper;
    MoveL Offs(pOrigin,155.6,107.2,0.0),vDraw,z1,tPen\WObj:=wPaper;
    MoveL Offs(pOrigin,156.2,107.2,0.0),vDraw,z1,tPen\WObj:=wPaper;
  ENDPROC

  PROC Part78()
    MoveL Offs(pOrigin,156.4,107.0,0.0),vDraw,z1,tPen\WObj:=wPaper;
    MoveL Offs(pOrigin,156.7,107.0,0.0),vDraw,z1,tPen\WObj:=wPaper;
    MoveL Offs(pOrigin,157.3,106.6,0.0),vDraw,z1,tPen\WObj:=wPaper;
    MoveL Offs(pOrigin,157.7,106.6,0.0),vDraw,z1,tPen\WObj:=wPaper;
    MoveL Offs(pOrigin,157.9,106.4,0.0),vDraw,z1,tPen\WObj:=wPaper;
    MoveL Offs(pOrigin,158.8,106.2,0.0),vDraw,z1,tPen\WObj:=wPaper;
    MoveL Offs(pOrigin,159.4,105.9,0.0),vDraw,z1,tPen\WObj:=wPaper;
    MoveL Offs(pOrigin,159.8,105.9,0.0),vDraw,z1,tPen\WObj:=wPaper;
    MoveL Offs(pOrigin,160.3,105.5,0.0),vDraw,z1,tPen\WObj:=wPaper;
    MoveL Offs(pOrigin,160.7,105.5,0.0),vDraw,z1,tPen\WObj:=wPaper;
    MoveL Offs(pOrigin,161.6,104.9,0.0),vDraw,z1,tPen\WObj:=wPaper;
    MoveL Offs(pOrigin,162.0,104.9,0.0),vDraw,z1,tPen\WObj:=wPaper;
    MoveL Offs(pOrigin,163.0,104.4,0.0),vDraw,z1,tPen\WObj:=wPaper;
    MoveL Offs(pOrigin,163.3,104.4,0.0),vDraw,z1,tPen\WObj:=wPaper;
    MoveL Offs(pOrigin,164.3,103.8,0.0),vDraw,z1,tPen\WObj:=wPaper;
    MoveL Offs(pOrigin,164.7,103.8,0.0),vDraw,z1,tPen\WObj:=wPaper;
    MoveL Offs(pOrigin,166.0,103.0,0.0),vDraw,z1,tPen\WObj:=wPaper;
    MoveL Offs(pOrigin,166.4,103.0,0.0),vDraw,z1,tPen\WObj:=wPaper;
    MoveL Offs(pOrigin,166.9,102.7,0.0),vDraw,z1,tPen\WObj:=wPaper;
    MoveL Offs(pOrigin,167.9,102.5,0.0),vDraw,z1,tPen\WObj:=wPaper;
    MoveL Offs(pOrigin,168.4,102.1,0.0),vDraw,z1,tPen\WObj:=wPaper;
    MoveL Offs(pOrigin,168.8,102.1,0.0),vDraw,z1,tPen\WObj:=wPaper;
    MoveL Offs(pOrigin,169.0,101.9,0.0),vDraw,z1,tPen\WObj:=wPaper;
    MoveL Offs(pOrigin,169.4,101.9,0.0),vDraw,z1,tPen\WObj:=wPaper;
    MoveL Offs(pOrigin,169.6,101.7,0.0),vDraw,z1,tPen\WObj:=wPaper;
    MoveL Offs(pOrigin,170.0,101.7,0.0),vDraw,z1,tPen\WObj:=wPaper;
    MoveL Offs(pOrigin,170.1,101.5,0.0),vDraw,z1,tPen\WObj:=wPaper;
    MoveL Offs(pOrigin,170.5,101.5,0.0),vDraw,z1,tPen\WObj:=wPaper;
    MoveL Offs(pOrigin,170.7,101.3,0.0),vDraw,z1,tPen\WObj:=wPaper;
    MoveL Offs(pOrigin,171.1,101.3,0.0),vDraw,z1,tPen\WObj:=wPaper;
    MoveL Offs(pOrigin,171.3,101.1,0.0),vDraw,z1,tPen\WObj:=wPaper;
    MoveL Offs(pOrigin,171.8,101.1,0.0),vDraw,z1,tPen\WObj:=wPaper;
    MoveL Offs(pOrigin,172.0,101.0,0.0),vDraw,z1,tPen\WObj:=wPaper;
    MoveL Offs(pOrigin,172.4,101.0,0.0),vDraw,z1,tPen\WObj:=wPaper;
    MoveL Offs(pOrigin,172.6,100.8,0.0),vDraw,z1,tPen\WObj:=wPaper;
    MoveL Offs(pOrigin,173.2,100.8,0.0),vDraw,z1,tPen\WObj:=wPaper;
    MoveL Offs(pOrigin,173.4,100.6,0.0),vDraw,z1,tPen\WObj:=wPaper;
    MoveL Offs(pOrigin,173.7,100.6,0.0),vDraw,z1,tPen\WObj:=wPaper;
    MoveL Offs(pOrigin,173.9,100.4,0.0),vDraw,z1,tPen\WObj:=wPaper;
    MoveL Offs(pOrigin,174.3,100.4,0.0),vDraw,z1,tPen\WObj:=wPaper;
    MoveL Offs(pOrigin,174.5,100.2,0.0),vDraw,z1,tPen\WObj:=wPaper;
    MoveL Offs(pOrigin,175.1,100.2,0.0),vDraw,z1,tPen\WObj:=wPaper;
    MoveL Offs(pOrigin,175.2,100.0,0.0),vDraw,z1,tPen\WObj:=wPaper;
    MoveL Offs(pOrigin,175.8,100.0,0.0),vDraw,z1,tPen\WObj:=wPaper;
    MoveL Offs(pOrigin,176.0,99.8,0.0),vDraw,z1,tPen\WObj:=wPaper;
    MoveL Offs(pOrigin,176.4,99.8,0.0),vDraw,z1,tPen\WObj:=wPaper;
    MoveL Offs(pOrigin,176.6,99.6,0.0),vDraw,z1,tPen\WObj:=wPaper;
    MoveL Offs(pOrigin,177.1,99.6,0.0),vDraw,z1,tPen\WObj:=wPaper;
    MoveL Offs(pOrigin,177.3,99.4,0.0),vDraw,z1,tPen\WObj:=wPaper;
    MoveL Offs(pOrigin,177.9,99.4,0.0),vDraw,z1,tPen\WObj:=wPaper;
    MoveL Offs(pOrigin,178.1,99.3,0.0),vDraw,z1,tPen\WObj:=wPaper;
    MoveL Offs(pOrigin,178.5,99.3,0.0),vDraw,z1,tPen\WObj:=wPaper;
    MoveL Offs(pOrigin,178.6,99.1,0.0),vDraw,z1,tPen\WObj:=wPaper;
    MoveL Offs(pOrigin,179.2,99.1,0.0),vDraw,z1,tPen\WObj:=wPaper;
    MoveL Offs(pOrigin,179.4,98.9,0.0),vDraw,z1,tPen\WObj:=wPaper;
    MoveL Offs(pOrigin,180.0,98.9,0.0),vDraw,z1,tPen\WObj:=wPaper;
    MoveL Offs(pOrigin,180.2,98.7,0.0),vDraw,z1,tPen\WObj:=wPaper;
    MoveL Offs(pOrigin,180.7,98.7,0.0),vDraw,z1,tPen\WObj:=wPaper;
    MoveL Offs(pOrigin,180.9,98.5,0.0),vDraw,z1,tPen\WObj:=wPaper;
    MoveL Offs(pOrigin,181.5,98.5,0.0),vDraw,z1,tPen\WObj:=wPaper;
    MoveL Offs(pOrigin,181.7,98.3,0.0),vDraw,z1,tPen\WObj:=wPaper;
    MoveL Offs(pOrigin,182.2,98.3,0.0),vDraw,z1,tPen\WObj:=wPaper;
    MoveL Offs(pOrigin,182.4,98.1,0.0),vDraw,z1,tPen\WObj:=wPaper;
    MoveL Offs(pOrigin,182.8,98.1,0.0),vDraw,z1,tPen\WObj:=wPaper;
    MoveL Offs(pOrigin,183.0,97.9,0.0),vDraw,z1,tPen\WObj:=wPaper;
    MoveL Offs(pOrigin,183.6,97.9,0.0),vDraw,z1,tPen\WObj:=wPaper;
    MoveL Offs(pOrigin,183.7,97.7,0.0),vDraw,z1,tPen\WObj:=wPaper;
    MoveL Offs(pOrigin,184.1,97.7,0.0),vDraw,z1,tPen\WObj:=wPaper;
    MoveL Offs(pOrigin,184.7,97.4,0.0),vDraw,z1,tPen\WObj:=wPaper;
    MoveL Offs(pOrigin,184.7,97.0,0.0),vDraw,z1,tPen\WObj:=wPaper;
    MoveL Offs(pOrigin,184.1,96.2,0.0),vDraw,z1,tPen\WObj:=wPaper;
    MoveL Offs(pOrigin,184.1,96.0,0.0),vDraw,z1,tPen\WObj:=wPaper;
    MoveL Offs(pOrigin,183.7,95.7,0.0),vDraw,z1,tPen\WObj:=wPaper;
    MoveL Offs(pOrigin,183.7,95.5,0.0),vDraw,z1,tPen\WObj:=wPaper;
    MoveL Offs(pOrigin,183.2,94.5,0.0),vDraw,z1,tPen\WObj:=wPaper;
    MoveL Offs(pOrigin,183.2,94.2,0.0),vDraw,z1,tPen\WObj:=wPaper;
    MoveL Offs(pOrigin,182.8,93.6,0.0),vDraw,z1,tPen\WObj:=wPaper;
    MoveL Offs(pOrigin,182.8,93.2,0.0),vDraw,z1,tPen\WObj:=wPaper;
    MoveL Offs(pOrigin,182.6,93.0,0.0),vDraw,z1,tPen\WObj:=wPaper;
    MoveL Offs(pOrigin,182.6,92.6,0.0),vDraw,z1,tPen\WObj:=wPaper;
    MoveL Offs(pOrigin,182.2,92.1,0.0),vDraw,z1,tPen\WObj:=wPaper;
    MoveL Offs(pOrigin,182.2,91.7,0.0),vDraw,z1,tPen\WObj:=wPaper;
    MoveL Offs(pOrigin,182.0,91.5,0.0),vDraw,z1,tPen\WObj:=wPaper;
    MoveL Offs(pOrigin,182.0,91.1,0.0),vDraw,z1,tPen\WObj:=wPaper;
    MoveL Offs(pOrigin,181.9,90.9,0.0),vDraw,z1,tPen\WObj:=wPaper;
    MoveL Offs(pOrigin,181.9,90.6,0.0),vDraw,z1,tPen\WObj:=wPaper;
    MoveL Offs(pOrigin,181.7,90.4,0.0),vDraw,z1,tPen\WObj:=wPaper;
    MoveL Offs(pOrigin,181.7,90.0,0.0),vDraw,z1,tPen\WObj:=wPaper;
    MoveL Offs(pOrigin,181.5,89.8,0.0),vDraw,z1,tPen\WObj:=wPaper;
    MoveL Offs(pOrigin,181.5,89.2,0.0),vDraw,z1,tPen\WObj:=wPaper;
    MoveL Offs(pOrigin,181.3,89.1,0.0),vDraw,z1,tPen\WObj:=wPaper;
    MoveL Offs(pOrigin,181.3,88.7,0.0),vDraw,z1,tPen\WObj:=wPaper;
    MoveL Offs(pOrigin,181.1,88.5,0.0),vDraw,z1,tPen\WObj:=wPaper;
    MoveL Offs(pOrigin,181.1,88.1,0.0),vDraw,z1,tPen\WObj:=wPaper;
    MoveL Offs(pOrigin,180.9,87.9,0.0),vDraw,z1,tPen\WObj:=wPaper;
    MoveL Offs(pOrigin,180.9,87.4,0.0),vDraw,z1,tPen\WObj:=wPaper;
    MoveL Offs(pOrigin,180.7,87.2,0.0),vDraw,z1,tPen\WObj:=wPaper;
    MoveL Offs(pOrigin,180.7,86.8,0.0),vDraw,z1,tPen\WObj:=wPaper;
    MoveL Offs(pOrigin,180.5,86.6,0.0),vDraw,z1,tPen\WObj:=wPaper;
    MoveL Offs(pOrigin,180.5,86.0,0.0),vDraw,z1,tPen\WObj:=wPaper;
    MoveL Offs(pOrigin,180.3,85.8,0.0),vDraw,z1,tPen\WObj:=wPaper;
    MoveL Offs(pOrigin,180.3,85.5,0.0),vDraw,z1,tPen\WObj:=wPaper;
    MoveL Offs(pOrigin,180.2,85.3,0.0),vDraw,z1,tPen\WObj:=wPaper;
    MoveL Offs(pOrigin,180.2,84.7,0.0),vDraw,z1,tPen\WObj:=wPaper;
    MoveL Offs(pOrigin,180.0,84.5,0.0),vDraw,z1,tPen\WObj:=wPaper;
    MoveL Offs(pOrigin,180.0,84.1,0.0),vDraw,z1,tPen\WObj:=wPaper;
    MoveL Offs(pOrigin,179.8,84.0,0.0),vDraw,z1,tPen\WObj:=wPaper;
    MoveL Offs(pOrigin,179.8,83.4,0.0),vDraw,z1,tPen\WObj:=wPaper;
    MoveL Offs(pOrigin,179.6,83.2,0.0),vDraw,z1,tPen\WObj:=wPaper;
    MoveL Offs(pOrigin,179.6,82.6,0.0),vDraw,z1,tPen\WObj:=wPaper;
    MoveL Offs(pOrigin,179.4,82.4,0.0),vDraw,z1,tPen\WObj:=wPaper;
    MoveL Offs(pOrigin,179.4,82.1,0.0),vDraw,z1,tPen\WObj:=wPaper;
    MoveL Offs(pOrigin,179.2,81.9,0.0),vDraw,z1,tPen\WObj:=wPaper;
    MoveL Offs(pOrigin,179.2,81.3,0.0),vDraw,z1,tPen\WObj:=wPaper;
    MoveL Offs(pOrigin,179.0,81.1,0.0),vDraw,z1,tPen\WObj:=wPaper;
    MoveL Offs(pOrigin,179.0,80.6,0.0),vDraw,z1,tPen\WObj:=wPaper;
    MoveL Offs(pOrigin,178.8,80.4,0.0),vDraw,z1,tPen\WObj:=wPaper;
    MoveL Offs(pOrigin,178.8,79.8,0.0),vDraw,z1,tPen\WObj:=wPaper;
    MoveL Offs(pOrigin,178.6,79.6,0.0),vDraw,z1,tPen\WObj:=wPaper;
    MoveL Offs(pOrigin,178.6,79.0,0.0),vDraw,z1,tPen\WObj:=wPaper;
  ENDPROC

  PROC Part79()
    MoveL Offs(pOrigin,178.5,78.9,0.0),vDraw,z1,tPen\WObj:=wPaper;
    MoveL Offs(pOrigin,178.5,78.3,0.0),vDraw,z1,tPen\WObj:=wPaper;
    MoveL Offs(pOrigin,178.3,78.1,0.0),vDraw,z1,tPen\WObj:=wPaper;
    MoveL Offs(pOrigin,178.3,77.5,0.0),vDraw,z1,tPen\WObj:=wPaper;
    MoveL Offs(pOrigin,178.1,77.3,0.0),vDraw,z1,tPen\WObj:=wPaper;
    MoveL Offs(pOrigin,178.1,76.8,0.0),vDraw,z1,tPen\WObj:=wPaper;
    MoveL Offs(pOrigin,177.9,76.6,0.0),vDraw,z1,tPen\WObj:=wPaper;
    MoveL Offs(pOrigin,177.9,76.0,0.0),vDraw,z1,tPen\WObj:=wPaper;
    MoveL Offs(pOrigin,177.7,75.8,0.0),vDraw,z1,tPen\WObj:=wPaper;
    MoveL Offs(pOrigin,177.7,75.3,0.0),vDraw,z1,tPen\WObj:=wPaper;
    MoveL Offs(pOrigin,177.5,75.1,0.0),vDraw,z1,tPen\WObj:=wPaper;
    MoveL Offs(pOrigin,177.5,74.5,0.0),vDraw,z1,tPen\WObj:=wPaper;
    MoveL Offs(pOrigin,177.3,74.3,0.0),vDraw,z1,tPen\WObj:=wPaper;
    MoveL Offs(pOrigin,177.3,73.8,0.0),vDraw,z1,tPen\WObj:=wPaper;
    MoveL Offs(pOrigin,177.1,73.6,0.0),vDraw,z1,tPen\WObj:=wPaper;
    MoveL Offs(pOrigin,177.1,72.8,0.0),vDraw,z1,tPen\WObj:=wPaper;
    MoveL Offs(pOrigin,176.9,72.6,0.0),vDraw,z1,tPen\WObj:=wPaper;
    MoveL Offs(pOrigin,176.9,72.1,0.0),vDraw,z1,tPen\WObj:=wPaper;
    MoveL Offs(pOrigin,176.8,71.9,0.0),vDraw,z1,tPen\WObj:=wPaper;
    MoveL Offs(pOrigin,176.8,71.1,0.0),vDraw,z1,tPen\WObj:=wPaper;
    MoveL Offs(pOrigin,176.6,70.9,0.0),vDraw,z1,tPen\WObj:=wPaper;
    MoveL Offs(pOrigin,176.6,70.4,0.0),vDraw,z1,tPen\WObj:=wPaper;
    MoveL Offs(pOrigin,176.4,70.2,0.0),vDraw,z1,tPen\WObj:=wPaper;
    MoveL Offs(pOrigin,176.4,69.6,0.0),vDraw,z1,tPen\WObj:=wPaper;
    MoveL Offs(pOrigin,176.2,69.4,0.0),vDraw,z1,tPen\WObj:=wPaper;
    MoveL Offs(pOrigin,176.2,68.7,0.0),vDraw,z1,tPen\WObj:=wPaper;
    MoveL Offs(pOrigin,176.0,68.5,0.0),vDraw,z1,tPen\WObj:=wPaper;
    MoveL Offs(pOrigin,176.0,67.7,0.0),vDraw,z1,tPen\WObj:=wPaper;
    MoveL Offs(pOrigin,175.8,67.5,0.0),vDraw,z1,tPen\WObj:=wPaper;
    MoveL Offs(pOrigin,175.8,66.8,0.0),vDraw,z1,tPen\WObj:=wPaper;
    MoveL Offs(pOrigin,175.6,66.6,0.0),vDraw,z1,tPen\WObj:=wPaper;
    MoveL Offs(pOrigin,175.6,65.8,0.0),vDraw,z1,tPen\WObj:=wPaper;
    MoveL Offs(pOrigin,175.4,65.6,0.0),vDraw,z1,tPen\WObj:=wPaper;
    MoveL Offs(pOrigin,175.4,64.9,0.0),vDraw,z1,tPen\WObj:=wPaper;
    MoveL Offs(pOrigin,175.2,64.7,0.0),vDraw,z1,tPen\WObj:=wPaper;
    MoveL Offs(pOrigin,175.2,63.7,0.0),vDraw,z1,tPen\WObj:=wPaper;
    MoveL Offs(pOrigin,175.1,63.6,0.0),vDraw,z1,tPen\WObj:=wPaper;
    MoveL Offs(pOrigin,175.1,62.8,0.0),vDraw,z1,tPen\WObj:=wPaper;
    MoveL Offs(pOrigin,174.9,62.6,0.0),vDraw,z1,tPen\WObj:=wPaper;
    MoveL Offs(pOrigin,174.9,61.9,0.0),vDraw,z1,tPen\WObj:=wPaper;
    MoveL Offs(pOrigin,174.7,61.7,0.0),vDraw,z1,tPen\WObj:=wPaper;
    MoveL Offs(pOrigin,174.7,60.9,0.0),vDraw,z1,tPen\WObj:=wPaper;
    MoveL Offs(pOrigin,174.5,60.7,0.0),vDraw,z1,tPen\WObj:=wPaper;
    MoveL Offs(pOrigin,174.5,60.2,0.0),vDraw,z1,tPen\WObj:=wPaper;
    MoveL Offs(pOrigin,174.3,60.0,0.0),vDraw,z1,tPen\WObj:=wPaper;
    MoveL Offs(pOrigin,174.3,59.4,0.0),vDraw,z1,tPen\WObj:=wPaper;
    MoveL Offs(pOrigin,174.1,59.2,0.0),vDraw,z1,tPen\WObj:=wPaper;
    MoveL Offs(pOrigin,174.1,58.6,0.0),vDraw,z1,tPen\WObj:=wPaper;
    MoveL Offs(pOrigin,173.9,58.5,0.0),vDraw,z1,tPen\WObj:=wPaper;
    MoveL Offs(pOrigin,173.9,57.9,0.0),vDraw,z1,tPen\WObj:=wPaper;
    MoveL Offs(pOrigin,173.7,57.7,0.0),vDraw,z1,tPen\WObj:=wPaper;
    MoveL Offs(pOrigin,173.7,57.3,0.0),vDraw,z1,tPen\WObj:=wPaper;
    MoveL Offs(pOrigin,173.5,57.1,0.0),vDraw,z1,tPen\WObj:=wPaper;
    MoveL Offs(pOrigin,173.5,56.8,0.0),vDraw,z1,tPen\WObj:=wPaper;
    MoveL Offs(pOrigin,173.4,56.6,0.0),vDraw,z1,tPen\WObj:=wPaper;
    MoveL Offs(pOrigin,173.4,56.0,0.0),vDraw,z1,tPen\WObj:=wPaper;
    MoveL Offs(pOrigin,173.2,55.8,0.0),vDraw,z1,tPen\WObj:=wPaper;
    MoveL Offs(pOrigin,173.2,55.4,0.0),vDraw,z1,tPen\WObj:=wPaper;
    MoveL Offs(pOrigin,173.0,55.2,0.0),vDraw,z1,tPen\WObj:=wPaper;
    MoveL Offs(pOrigin,173.0,54.9,0.0),vDraw,z1,tPen\WObj:=wPaper;
    MoveL Offs(pOrigin,172.8,54.7,0.0),vDraw,z1,tPen\WObj:=wPaper;
    MoveL Offs(pOrigin,172.8,54.3,0.0),vDraw,z1,tPen\WObj:=wPaper;
    MoveL Offs(pOrigin,172.6,54.1,0.0),vDraw,z1,tPen\WObj:=wPaper;
    MoveL Offs(pOrigin,172.6,53.7,0.0),vDraw,z1,tPen\WObj:=wPaper;
    MoveL Offs(pOrigin,172.4,53.5,0.0),vDraw,z1,tPen\WObj:=wPaper;
    MoveL Offs(pOrigin,172.2,52.6,0.0),vDraw,z1,tPen\WObj:=wPaper;
    MoveL Offs(pOrigin,171.8,52.0,0.0),vDraw,z1,tPen\WObj:=wPaper;
    MoveL Offs(pOrigin,171.7,51.1,0.0),vDraw,z1,tPen\WObj:=wPaper;
    MoveL Offs(pOrigin,171.3,50.5,0.0),vDraw,z1,tPen\WObj:=wPaper;
    MoveL Offs(pOrigin,171.1,49.6,0.0),vDraw,z1,tPen\WObj:=wPaper;
    MoveL Offs(pOrigin,170.7,49.0,0.0),vDraw,z1,tPen\WObj:=wPaper;
    MoveL Offs(pOrigin,170.7,48.6,0.0),vDraw,z1,tPen\WObj:=wPaper;
    MoveL Offs(pOrigin,170.1,47.7,0.0),vDraw,z1,tPen\WObj:=wPaper;
    MoveL Offs(pOrigin,170.0,46.7,0.0),vDraw,z1,tPen\WObj:=wPaper;
    MoveL Offs(pOrigin,169.4,45.8,0.0),vDraw,z1,tPen\WObj:=wPaper;
    MoveL Offs(pOrigin,169.4,45.4,0.0),vDraw,z1,tPen\WObj:=wPaper;
    MoveL Offs(pOrigin,169.0,44.9,0.0),vDraw,z1,tPen\WObj:=wPaper;
    MoveL Offs(pOrigin,169.0,44.5,0.0),vDraw,z1,tPen\WObj:=wPaper;
    MoveL Offs(pOrigin,168.8,44.3,0.0),vDraw,z1,tPen\WObj:=wPaper;
    MoveL Offs(pOrigin,168.8,44.1,0.0),vDraw,z1,tPen\WObj:=wPaper;
    MoveL Offs(pOrigin,168.4,43.5,0.0),vDraw,z1,tPen\WObj:=wPaper;
    MoveL Offs(pOrigin,168.4,43.2,0.0),vDraw,z1,tPen\WObj:=wPaper;
    MoveL Offs(pOrigin,168.1,42.6,0.0),vDraw,z1,tPen\WObj:=wPaper;
    MoveL Offs(pOrigin,168.1,42.2,0.0),vDraw,z1,tPen\WObj:=wPaper;
    MoveL Offs(pOrigin,168.1,42.4,0.0),vDraw,z1,tPen\WObj:=wPaper;
    MoveL Offs(pOrigin,168.6,43.2,0.0),vDraw,z1,tPen\WObj:=wPaper;
    MoveL Offs(pOrigin,168.6,43.3,0.0),vDraw,z1,tPen\WObj:=wPaper;
    MoveL Offs(pOrigin,168.8,43.5,0.0),vDraw,z1,tPen\WObj:=wPaper;
    MoveL Offs(pOrigin,168.8,43.9,0.0),vDraw,z1,tPen\WObj:=wPaper;
    MoveL Offs(pOrigin,169.2,44.3,0.0),vDraw,z1,tPen\WObj:=wPaper;
    MoveL Offs(pOrigin,169.2,44.7,0.0),vDraw,z1,tPen\WObj:=wPaper;
    MoveL Offs(pOrigin,170.3,46.7,0.0),vDraw,z1,tPen\WObj:=wPaper;
    MoveL Offs(pOrigin,170.3,47.1,0.0),vDraw,z1,tPen\WObj:=wPaper;
    MoveL Offs(pOrigin,170.5,47.3,0.0),vDraw,z1,tPen\WObj:=wPaper;
    MoveL Offs(pOrigin,170.5,47.5,0.0),vDraw,z1,tPen\WObj:=wPaper;
    MoveL Offs(pOrigin,170.9,48.1,0.0),vDraw,z1,tPen\WObj:=wPaper;
    MoveL Offs(pOrigin,170.9,48.4,0.0),vDraw,z1,tPen\WObj:=wPaper;
    MoveL Offs(pOrigin,171.5,49.4,0.0),vDraw,z1,tPen\WObj:=wPaper;
    MoveL Offs(pOrigin,171.5,49.8,0.0),vDraw,z1,tPen\WObj:=wPaper;
    MoveL Offs(pOrigin,171.8,50.3,0.0),vDraw,z1,tPen\WObj:=wPaper;
    MoveL Offs(pOrigin,171.8,50.7,0.0),vDraw,z1,tPen\WObj:=wPaper;
    MoveL Offs(pOrigin,172.2,51.3,0.0),vDraw,z1,tPen\WObj:=wPaper;
    MoveL Offs(pOrigin,172.2,51.7,0.0),vDraw,z1,tPen\WObj:=wPaper;
    MoveL Offs(pOrigin,172.8,52.6,0.0),vDraw,z1,tPen\WObj:=wPaper;
    MoveL Offs(pOrigin,173.0,52.4,0.0),vDraw,z1,tPen\WObj:=wPaper;
    MoveL Offs(pOrigin,173.0,51.8,0.0),vDraw,z1,tPen\WObj:=wPaper;
    MoveL Offs(pOrigin,172.8,51.7,0.0),vDraw,z1,tPen\WObj:=wPaper;
    MoveL Offs(pOrigin,172.8,51.1,0.0),vDraw,z1,tPen\WObj:=wPaper;
    MoveL Offs(pOrigin,172.6,50.9,0.0),vDraw,z1,tPen\WObj:=wPaper;
    MoveL Offs(pOrigin,172.6,50.3,0.0),vDraw,z1,tPen\WObj:=wPaper;
    MoveL Offs(pOrigin,172.4,50.1,0.0),vDraw,z1,tPen\WObj:=wPaper;
    MoveL Offs(pOrigin,172.4,49.8,0.0),vDraw,z1,tPen\WObj:=wPaper;
    MoveL Offs(pOrigin,172.2,49.6,0.0),vDraw,z1,tPen\WObj:=wPaper;
    MoveL Offs(pOrigin,172.2,49.2,0.0),vDraw,z1,tPen\WObj:=wPaper;
    MoveL Offs(pOrigin,172.0,49.0,0.0),vDraw,z1,tPen\WObj:=wPaper;
    MoveL Offs(pOrigin,172.0,48.4,0.0),vDraw,z1,tPen\WObj:=wPaper;
    MoveL Offs(pOrigin,171.8,48.3,0.0),vDraw,z1,tPen\WObj:=wPaper;
    MoveL Offs(pOrigin,171.8,47.9,0.0),vDraw,z1,tPen\WObj:=wPaper;
    MoveL Offs(pOrigin,171.7,47.7,0.0),vDraw,z1,tPen\WObj:=wPaper;
    MoveL Offs(pOrigin,171.5,46.7,0.0),vDraw,z1,tPen\WObj:=wPaper;
  ENDPROC

  PROC Part80()
    MoveL Offs(pOrigin,171.1,46.2,0.0),vDraw,z1,tPen\WObj:=wPaper;
    MoveL Offs(pOrigin,170.9,45.2,0.0),vDraw,z1,tPen\WObj:=wPaper;
    MoveL Offs(pOrigin,170.5,44.7,0.0),vDraw,z1,tPen\WObj:=wPaper;
    MoveL Offs(pOrigin,170.5,44.3,0.0),vDraw,z1,tPen\WObj:=wPaper;
    MoveL Offs(pOrigin,170.0,43.3,0.0),vDraw,z1,tPen\WObj:=wPaper;
    MoveL Offs(pOrigin,170.0,43.0,0.0),vDraw,z1,tPen\WObj:=wPaper;
    MoveL Offs(pOrigin,169.4,42.0,0.0),vDraw,z1,tPen\WObj:=wPaper;
    MoveL Offs(pOrigin,169.4,41.6,0.0),vDraw,z1,tPen\WObj:=wPaper;
    MoveL Offs(pOrigin,169.2,41.5,0.0),vDraw,z1,tPen\WObj:=wPaper;
    MoveL Offs(pOrigin,168.8,40.5,0.0),vDraw,z1,tPen\WObj:=wPaper;
    MoveL Offs(pOrigin,168.4,40.1,0.0),vDraw,z1,tPen\WObj:=wPaper;
    MoveL Offs(pOrigin,168.1,40.1,0.0),vDraw,z1,tPen\WObj:=wPaper;
    MoveL Offs(pOrigin,167.9,39.9,0.0),vDraw,z1,tPen\WObj:=wPaper;
    MoveL Offs(pOrigin,166.7,39.9,0.0),vDraw,z1,tPen\WObj:=wPaper;
    MoveL Offs(pOrigin,166.6,39.8,0.0),vDraw,z1,tPen\WObj:=wPaper;
    MoveL Offs(pOrigin,165.6,39.8,0.0),vDraw,z1,tPen\WObj:=wPaper;
    MoveL Offs(pOrigin,165.4,39.6,0.0),vDraw,z1,tPen\WObj:=wPaper;
    MoveL Offs(pOrigin,164.7,39.6,0.0),vDraw,z1,tPen\WObj:=wPaper;
    MoveL Offs(pOrigin,164.5,39.4,0.0),vDraw,z1,tPen\WObj:=wPaper;
    MoveL Offs(pOrigin,163.5,39.4,0.0),vDraw,z1,tPen\WObj:=wPaper;
    MoveL Offs(pOrigin,163.3,39.2,0.0),vDraw,z1,tPen\WObj:=wPaper;
    MoveL Offs(pOrigin,162.6,39.2,0.0),vDraw,z1,tPen\WObj:=wPaper;
    MoveL Offs(pOrigin,162.4,39.0,0.0),vDraw,z1,tPen\WObj:=wPaper;
    MoveL Offs(pOrigin,161.6,39.0,0.0),vDraw,z1,tPen\WObj:=wPaper;
    MoveL Offs(pOrigin,161.5,38.8,0.0),vDraw,z1,tPen\WObj:=wPaper;
    MoveL Offs(pOrigin,160.9,38.8,0.0),vDraw,z1,tPen\WObj:=wPaper;
    MoveL Offs(pOrigin,160.7,38.6,0.0),vDraw,z1,tPen\WObj:=wPaper;
    MoveL Offs(pOrigin,160.1,38.6,0.0),vDraw,z1,tPen\WObj:=wPaper;
    MoveL Offs(pOrigin,159.9,38.4,0.0),vDraw,z1,tPen\WObj:=wPaper;
    MoveL Offs(pOrigin,159.4,38.4,0.0),vDraw,z1,tPen\WObj:=wPaper;
    MoveL Offs(pOrigin,159.2,38.2,0.0),vDraw,z1,tPen\WObj:=wPaper;
    MoveL Offs(pOrigin,158.8,38.2,0.0),vDraw,z1,tPen\WObj:=wPaper;
    MoveL Offs(pOrigin,158.6,38.1,0.0),vDraw,z1,tPen\WObj:=wPaper;
    MoveL Offs(pOrigin,157.7,37.9,0.0),vDraw,z1,tPen\WObj:=wPaper;
    MoveL Offs(pOrigin,157.5,37.7,0.0),vDraw,z1,tPen\WObj:=wPaper;
    MoveL Offs(pOrigin,157.3,37.7,0.0),vDraw,z1,tPen\WObj:=wPaper;
    MoveL Offs(pOrigin,157.1,37.5,0.0),vDraw,z1,tPen\WObj:=wPaper;
    MoveL Offs(pOrigin,155.8,36.9,0.0),vDraw,z1,tPen\WObj:=wPaper;
    MoveL Offs(pOrigin,154.8,36.2,0.0),vDraw,z1,tPen\WObj:=wPaper;
    MoveL Offs(pOrigin,154.3,36.2,0.0),vDraw,z1,tPen\WObj:=wPaper;
    MoveL Offs(pOrigin,154.1,36.0,0.0),vDraw,z1,tPen\WObj:=wPaper;
    MoveL Offs(pOrigin,153.3,36.0,0.0),vDraw,z1,tPen\WObj:=wPaper;
    MoveL Offs(pOrigin,153.1,35.8,0.0),vDraw,z1,tPen\WObj:=wPaper;
    MoveL Offs(pOrigin,152.6,35.8,0.0),vDraw,z1,tPen\WObj:=wPaper;
    MoveL Offs(pOrigin,152.4,35.6,0.0),vDraw,z1,tPen\WObj:=wPaper;
    MoveL Offs(pOrigin,151.4,35.4,0.0),vDraw,z1,tPen\WObj:=wPaper;
    MoveL Offs(pOrigin,150.9,35.0,0.0),vDraw,z1,tPen\WObj:=wPaper;
    MoveL Offs(pOrigin,150.5,35.0,0.0),vDraw,z1,tPen\WObj:=wPaper;
    MoveL Offs(pOrigin,150.3,34.8,0.0),vDraw,z1,tPen\WObj:=wPaper;
    MoveL Offs(pOrigin,150.1,34.8,0.0),vDraw,z1,tPen\WObj:=wPaper;
    MoveL Offs(pOrigin,149.0,33.9,0.0),vDraw,z1,tPen\WObj:=wPaper;
    MoveL Offs(pOrigin,148.6,33.9,0.0),vDraw,z1,tPen\WObj:=wPaper;
    MoveL Offs(pOrigin,148.4,34.1,0.0),vDraw,z1,tPen\WObj:=wPaper;
    MoveL Offs(pOrigin,148.0,34.1,0.0),vDraw,z1,tPen\WObj:=wPaper;
    MoveL Offs(pOrigin,147.5,34.5,0.0),vDraw,z1,tPen\WObj:=wPaper;
    MoveL Offs(pOrigin,146.5,34.7,0.0),vDraw,z1,tPen\WObj:=wPaper;
    MoveL Offs(pOrigin,146.0,35.0,0.0),vDraw,z1,tPen\WObj:=wPaper;
    MoveL Offs(pOrigin,145.6,35.0,0.0),vDraw,z1,tPen\WObj:=wPaper;
    MoveL Offs(pOrigin,145.4,35.2,0.0),vDraw,z1,tPen\WObj:=wPaper;
    MoveL Offs(pOrigin,144.8,35.4,0.0),vDraw,z1,tPen\WObj:=wPaper;
    MoveL Offs(pOrigin,144.5,35.8,0.0),vDraw,z1,tPen\WObj:=wPaper;
    MoveL Offs(pOrigin,144.3,35.8,0.0),vDraw,z1,tPen\WObj:=wPaper;
    MoveL Offs(pOrigin,143.9,36.2,0.0),vDraw,z1,tPen\WObj:=wPaper;
    MoveL Offs(pOrigin,143.7,36.2,0.0),vDraw,z1,tPen\WObj:=wPaper;
    MoveL Offs(pOrigin,143.1,36.7,0.0),vDraw,fine,tPen\WObj:=wPaper;
    MoveL Offs(pOrigin,143.1,36.7,15.0),vApproach,z5,tPen\WObj:=wPaper;
    MoveL Offs(pOrigin,152.0,34.7,15.0),vTravel,z5,tPen\WObj:=wPaper;
    MoveL Offs(pOrigin,152.0,34.7,0.0),vApproach,fine,tPen\WObj:=wPaper;
    MoveL Offs(pOrigin,152.2,34.8,0.0),vDraw,z1,tPen\WObj:=wPaper;
    MoveL Offs(pOrigin,152.6,34.8,0.0),vDraw,z1,tPen\WObj:=wPaper;
    MoveL Offs(pOrigin,152.8,35.0,0.0),vDraw,z1,tPen\WObj:=wPaper;
    MoveL Offs(pOrigin,153.3,35.0,0.0),vDraw,z1,tPen\WObj:=wPaper;
    MoveL Offs(pOrigin,153.5,35.2,0.0),vDraw,z1,tPen\WObj:=wPaper;
    MoveL Offs(pOrigin,154.1,35.2,0.0),vDraw,z1,tPen\WObj:=wPaper;
    MoveL Offs(pOrigin,154.3,35.4,0.0),vDraw,z1,tPen\WObj:=wPaper;
    MoveL Offs(pOrigin,155.0,35.4,0.0),vDraw,z1,tPen\WObj:=wPaper;
    MoveL Offs(pOrigin,155.2,35.6,0.0),vDraw,z1,tPen\WObj:=wPaper;
    MoveL Offs(pOrigin,156.2,35.6,0.0),vDraw,z1,tPen\WObj:=wPaper;
    MoveL Offs(pOrigin,156.4,35.8,0.0),vDraw,z1,tPen\WObj:=wPaper;
    MoveL Offs(pOrigin,157.3,35.8,0.0),vDraw,z1,tPen\WObj:=wPaper;
    MoveL Offs(pOrigin,157.5,36.0,0.0),vDraw,z1,tPen\WObj:=wPaper;
    MoveL Offs(pOrigin,158.4,36.0,0.0),vDraw,z1,tPen\WObj:=wPaper;
    MoveL Offs(pOrigin,158.6,36.2,0.0),vDraw,z1,tPen\WObj:=wPaper;
    MoveL Offs(pOrigin,160.9,36.2,0.0),vDraw,z1,tPen\WObj:=wPaper;
    MoveL Offs(pOrigin,161.1,36.0,0.0),vDraw,z1,tPen\WObj:=wPaper;
    MoveL Offs(pOrigin,161.6,36.0,0.0),vDraw,z1,tPen\WObj:=wPaper;
    MoveL Offs(pOrigin,161.8,35.8,0.0),vDraw,z1,tPen\WObj:=wPaper;
    MoveL Offs(pOrigin,162.8,35.6,0.0),vDraw,z1,tPen\WObj:=wPaper;
    MoveL Offs(pOrigin,163.0,35.4,0.0),vDraw,z1,tPen\WObj:=wPaper;
    MoveL Offs(pOrigin,163.2,35.4,0.0),vDraw,z1,tPen\WObj:=wPaper;
    MoveL Offs(pOrigin,163.3,35.2,0.0),vDraw,z1,tPen\WObj:=wPaper;
    MoveL Offs(pOrigin,163.5,35.2,0.0),vDraw,z1,tPen\WObj:=wPaper;
    MoveL Offs(pOrigin,163.7,35.0,0.0),vDraw,z1,tPen\WObj:=wPaper;
    MoveL Offs(pOrigin,165.0,34.5,0.0),vDraw,z1,tPen\WObj:=wPaper;
    MoveL Offs(pOrigin,165.4,34.1,0.0),vDraw,z1,tPen\WObj:=wPaper;
    MoveL Offs(pOrigin,165.6,34.1,0.0),vDraw,z1,tPen\WObj:=wPaper;
    MoveL Offs(pOrigin,166.0,33.7,0.0),vDraw,z1,tPen\WObj:=wPaper;
    MoveL Offs(pOrigin,166.2,33.7,0.0),vDraw,z1,tPen\WObj:=wPaper;
    MoveL Offs(pOrigin,166.6,33.3,0.0),vDraw,z1,tPen\WObj:=wPaper;
    MoveL Offs(pOrigin,166.7,33.3,0.0),vDraw,z1,tPen\WObj:=wPaper;
    MoveL Offs(pOrigin,167.7,32.4,0.0),vDraw,z1,tPen\WObj:=wPaper;
    MoveL Offs(pOrigin,167.9,32.4,0.0),vDraw,z1,tPen\WObj:=wPaper;
    MoveL Offs(pOrigin,169.8,30.5,0.0),vDraw,z1,tPen\WObj:=wPaper;
    MoveL Offs(pOrigin,169.8,30.3,0.0),vDraw,z1,tPen\WObj:=wPaper;
    MoveL Offs(pOrigin,170.7,29.4,0.0),vDraw,z1,tPen\WObj:=wPaper;
    MoveL Offs(pOrigin,170.7,29.2,0.0),vDraw,z1,tPen\WObj:=wPaper;
    MoveL Offs(pOrigin,171.1,28.8,0.0),vDraw,z1,tPen\WObj:=wPaper;
    MoveL Offs(pOrigin,171.1,28.6,0.0),vDraw,z1,tPen\WObj:=wPaper;
    MoveL Offs(pOrigin,172.0,27.5,0.0),vDraw,z1,tPen\WObj:=wPaper;
    MoveL Offs(pOrigin,172.2,26.9,0.0),vDraw,z1,tPen\WObj:=wPaper;
    MoveL Offs(pOrigin,172.6,26.5,0.0),vDraw,z1,tPen\WObj:=wPaper;
    MoveL Offs(pOrigin,172.8,26.0,0.0),vDraw,z1,tPen\WObj:=wPaper;
    MoveL Offs(pOrigin,173.2,25.6,0.0),vDraw,z1,tPen\WObj:=wPaper;
    MoveL Offs(pOrigin,173.2,25.4,0.0),vDraw,z1,tPen\WObj:=wPaper;
    MoveL Offs(pOrigin,173.7,24.5,0.0),vDraw,z1,tPen\WObj:=wPaper;
    MoveL Offs(pOrigin,173.7,21.8,0.0),vDraw,z1,tPen\WObj:=wPaper;
    MoveL Offs(pOrigin,173.5,21.6,0.0),vDraw,z1,tPen\WObj:=wPaper;
    MoveL Offs(pOrigin,173.5,21.2,0.0),vDraw,z1,tPen\WObj:=wPaper;
    MoveL Offs(pOrigin,173.4,21.1,0.0),vDraw,z1,tPen\WObj:=wPaper;
    MoveL Offs(pOrigin,173.2,20.1,0.0),vDraw,z1,tPen\WObj:=wPaper;
  ENDPROC

  PROC Part81()
    MoveL Offs(pOrigin,172.8,19.7,0.0),vDraw,z1,tPen\WObj:=wPaper;
    MoveL Offs(pOrigin,172.8,19.5,0.0),vDraw,z1,tPen\WObj:=wPaper;
    MoveL Offs(pOrigin,171.5,18.2,0.0),vDraw,z1,tPen\WObj:=wPaper;
    MoveL Offs(pOrigin,171.3,18.2,0.0),vDraw,z1,tPen\WObj:=wPaper;
    MoveL Offs(pOrigin,170.9,17.8,0.0),vDraw,z1,tPen\WObj:=wPaper;
    MoveL Offs(pOrigin,170.5,17.8,0.0),vDraw,z1,tPen\WObj:=wPaper;
    MoveL Offs(pOrigin,170.3,17.7,0.0),vDraw,z1,tPen\WObj:=wPaper;
    MoveL Offs(pOrigin,170.0,17.7,0.0),vDraw,z1,tPen\WObj:=wPaper;
    MoveL Offs(pOrigin,169.8,17.5,0.0),vDraw,z1,tPen\WObj:=wPaper;
    MoveL Offs(pOrigin,169.4,17.5,0.0),vDraw,z1,tPen\WObj:=wPaper;
    MoveL Offs(pOrigin,169.2,17.3,0.0),vDraw,z1,tPen\WObj:=wPaper;
    MoveL Offs(pOrigin,168.6,17.3,0.0),vDraw,z1,tPen\WObj:=wPaper;
    MoveL Offs(pOrigin,168.4,17.1,0.0),vDraw,z1,tPen\WObj:=wPaper;
    MoveL Offs(pOrigin,167.7,17.1,0.0),vDraw,z1,tPen\WObj:=wPaper;
    MoveL Offs(pOrigin,167.5,16.9,0.0),vDraw,z1,tPen\WObj:=wPaper;
    MoveL Offs(pOrigin,166.7,16.9,0.0),vDraw,z1,tPen\WObj:=wPaper;
    MoveL Offs(pOrigin,166.6,16.7,0.0),vDraw,z1,tPen\WObj:=wPaper;
    MoveL Offs(pOrigin,165.8,16.7,0.0),vDraw,z1,tPen\WObj:=wPaper;
    MoveL Offs(pOrigin,165.6,16.5,0.0),vDraw,z1,tPen\WObj:=wPaper;
    MoveL Offs(pOrigin,164.9,16.5,0.0),vDraw,z1,tPen\WObj:=wPaper;
    MoveL Offs(pOrigin,164.7,16.3,0.0),vDraw,z1,tPen\WObj:=wPaper;
    MoveL Offs(pOrigin,163.9,16.3,0.0),vDraw,z1,tPen\WObj:=wPaper;
    MoveL Offs(pOrigin,163.7,16.1,0.0),vDraw,z1,tPen\WObj:=wPaper;
    MoveL Offs(pOrigin,162.6,16.1,0.0),vDraw,z1,tPen\WObj:=wPaper;
    MoveL Offs(pOrigin,162.4,16.0,0.0),vDraw,z1,tPen\WObj:=wPaper;
    MoveL Offs(pOrigin,161.5,16.0,0.0),vDraw,z1,tPen\WObj:=wPaper;
    MoveL Offs(pOrigin,161.3,15.8,0.0),vDraw,z1,tPen\WObj:=wPaper;
    MoveL Offs(pOrigin,159.9,15.8,0.0),vDraw,z1,tPen\WObj:=wPaper;
    MoveL Offs(pOrigin,159.8,16.0,0.0),vDraw,z1,tPen\WObj:=wPaper;
    MoveL Offs(pOrigin,160.9,17.1,0.0),vDraw,z1,tPen\WObj:=wPaper;
    MoveL Offs(pOrigin,160.9,17.3,0.0),vDraw,z1,tPen\WObj:=wPaper;
    MoveL Offs(pOrigin,161.6,18.6,0.0),vDraw,z1,tPen\WObj:=wPaper;
    MoveL Offs(pOrigin,161.6,19.2,0.0),vDraw,z1,tPen\WObj:=wPaper;
    MoveL Offs(pOrigin,161.8,19.4,0.0),vDraw,z1,tPen\WObj:=wPaper;
    MoveL Offs(pOrigin,161.8,19.7,0.0),vDraw,z1,tPen\WObj:=wPaper;
    MoveL Offs(pOrigin,162.0,19.9,0.0),vDraw,z1,tPen\WObj:=wPaper;
    MoveL Offs(pOrigin,162.0,20.7,0.0),vDraw,z1,tPen\WObj:=wPaper;
    MoveL Offs(pOrigin,162.2,20.9,0.0),vDraw,z1,tPen\WObj:=wPaper;
    MoveL Offs(pOrigin,162.2,22.2,0.0),vDraw,z1,tPen\WObj:=wPaper;
    MoveL Offs(pOrigin,162.4,22.4,0.0),vDraw,z1,tPen\WObj:=wPaper;
    MoveL Offs(pOrigin,162.4,24.3,0.0),vDraw,z1,tPen\WObj:=wPaper;
    MoveL Offs(pOrigin,162.2,24.5,0.0),vDraw,z1,tPen\WObj:=wPaper;
    MoveL Offs(pOrigin,162.2,25.8,0.0),vDraw,z1,tPen\WObj:=wPaper;
    MoveL Offs(pOrigin,162.0,26.0,0.0),vDraw,z1,tPen\WObj:=wPaper;
    MoveL Offs(pOrigin,162.0,26.7,0.0),vDraw,z1,tPen\WObj:=wPaper;
    MoveL Offs(pOrigin,161.8,26.9,0.0),vDraw,z1,tPen\WObj:=wPaper;
    MoveL Offs(pOrigin,161.8,27.5,0.0),vDraw,z1,tPen\WObj:=wPaper;
    MoveL Offs(pOrigin,161.6,27.7,0.0),vDraw,z1,tPen\WObj:=wPaper;
    MoveL Offs(pOrigin,161.6,28.0,0.0),vDraw,z1,tPen\WObj:=wPaper;
    MoveL Offs(pOrigin,161.5,28.2,0.0),vDraw,z1,tPen\WObj:=wPaper;
    MoveL Offs(pOrigin,161.5,28.6,0.0),vDraw,z1,tPen\WObj:=wPaper;
    MoveL Offs(pOrigin,161.3,28.8,0.0),vDraw,z1,tPen\WObj:=wPaper;
    MoveL Offs(pOrigin,161.1,29.7,0.0),vDraw,z1,tPen\WObj:=wPaper;
    MoveL Offs(pOrigin,160.9,29.9,0.0),vDraw,z1,tPen\WObj:=wPaper;
    MoveL Offs(pOrigin,160.3,31.3,0.0),vDraw,z1,tPen\WObj:=wPaper;
    MoveL Offs(pOrigin,159.8,31.8,0.0),vDraw,z1,tPen\WObj:=wPaper;
    MoveL Offs(pOrigin,159.8,32.0,0.0),vDraw,z1,tPen\WObj:=wPaper;
    MoveL Offs(pOrigin,158.6,33.1,0.0),vDraw,z1,tPen\WObj:=wPaper;
    MoveL Offs(pOrigin,158.4,33.1,0.0),vDraw,z1,tPen\WObj:=wPaper;
    MoveL Offs(pOrigin,158.1,33.5,0.0),vDraw,z1,tPen\WObj:=wPaper;
    MoveL Offs(pOrigin,157.9,33.5,0.0),vDraw,z1,tPen\WObj:=wPaper;
    MoveL Offs(pOrigin,156.9,34.1,0.0),vDraw,z1,tPen\WObj:=wPaper;
    MoveL Offs(pOrigin,156.0,34.3,0.0),vDraw,z1,tPen\WObj:=wPaper;
    MoveL Offs(pOrigin,155.8,34.5,0.0),vDraw,z1,tPen\WObj:=wPaper;
    MoveL Offs(pOrigin,154.8,34.5,0.0),vDraw,z1,tPen\WObj:=wPaper;
    MoveL Offs(pOrigin,154.7,34.7,0.0),vDraw,z1,tPen\WObj:=wPaper;
    MoveL Offs(pOrigin,153.5,34.7,0.0),vDraw,z1,tPen\WObj:=wPaper;
    MoveL Offs(pOrigin,153.3,34.5,0.0),vDraw,z1,tPen\WObj:=wPaper;
    MoveL Offs(pOrigin,152.2,34.5,0.0),vDraw,z1,tPen\WObj:=wPaper;
    MoveL Offs(pOrigin,152.0,34.7,0.0),vDraw,fine,tPen\WObj:=wPaper;
    MoveL Offs(pOrigin,152.0,34.7,15.0),vApproach,z5,tPen\WObj:=wPaper;
    MoveL Offs(pOrigin,152.0,33.7,15.0),vTravel,z5,tPen\WObj:=wPaper;
    MoveL Offs(pOrigin,152.0,33.7,0.0),vApproach,fine,tPen\WObj:=wPaper;
    MoveL Offs(pOrigin,152.8,33.7,0.0),vDraw,z1,tPen\WObj:=wPaper;
    MoveL Offs(pOrigin,153.0,33.9,0.0),vDraw,z1,tPen\WObj:=wPaper;
    MoveL Offs(pOrigin,154.1,33.9,0.0),vDraw,z1,tPen\WObj:=wPaper;
    MoveL Offs(pOrigin,154.3,33.7,0.0),vDraw,z1,tPen\WObj:=wPaper;
    MoveL Offs(pOrigin,153.9,33.3,0.0),vDraw,z1,tPen\WObj:=wPaper;
    MoveL Offs(pOrigin,153.7,33.3,0.0),vDraw,z1,tPen\WObj:=wPaper;
    MoveL Offs(pOrigin,153.5,33.1,0.0),vDraw,z1,tPen\WObj:=wPaper;
    MoveL Offs(pOrigin,153.0,33.1,0.0),vDraw,z1,tPen\WObj:=wPaper;
    MoveL Offs(pOrigin,152.8,33.0,0.0),vDraw,z1,tPen\WObj:=wPaper;
    MoveL Offs(pOrigin,152.6,33.1,0.0),vDraw,z1,tPen\WObj:=wPaper;
    MoveL Offs(pOrigin,151.8,33.1,0.0),vDraw,z1,tPen\WObj:=wPaper;
    MoveL Offs(pOrigin,151.6,33.3,0.0),vDraw,z1,tPen\WObj:=wPaper;
    MoveL Offs(pOrigin,152.0,33.7,0.0),vDraw,fine,tPen\WObj:=wPaper;
    MoveL Offs(pOrigin,152.0,33.7,15.0),vApproach,z5,tPen\WObj:=wPaper;
    MoveL Offs(pOrigin,157.7,32.4,15.0),vTravel,z5,tPen\WObj:=wPaper;
    MoveL Offs(pOrigin,157.7,32.4,0.0),vApproach,fine,tPen\WObj:=wPaper;
    MoveL Offs(pOrigin,157.9,32.6,0.0),vDraw,z1,tPen\WObj:=wPaper;
    MoveL Offs(pOrigin,158.1,32.6,0.0),vDraw,z1,tPen\WObj:=wPaper;
    MoveL Offs(pOrigin,158.8,31.8,0.0),vDraw,z1,tPen\WObj:=wPaper;
    MoveL Offs(pOrigin,158.6,31.6,0.0),vDraw,z1,tPen\WObj:=wPaper;
    MoveL Offs(pOrigin,158.4,31.6,0.0),vDraw,z1,tPen\WObj:=wPaper;
    MoveL Offs(pOrigin,157.7,32.4,0.0),vDraw,fine,tPen\WObj:=wPaper;
    MoveL Offs(pOrigin,157.7,32.4,15.0),vApproach,z5,tPen\WObj:=wPaper;
    MoveL Offs(pOrigin,158.4,36.9,15.0),vTravel,z5,tPen\WObj:=wPaper;
    MoveL Offs(pOrigin,158.4,36.9,0.0),vApproach,fine,tPen\WObj:=wPaper;
    MoveL Offs(pOrigin,158.2,37.1,0.0),vDraw,z1,tPen\WObj:=wPaper;
    MoveL Offs(pOrigin,158.4,37.3,0.0),vDraw,z1,tPen\WObj:=wPaper;
    MoveL Offs(pOrigin,158.6,37.3,0.0),vDraw,z1,tPen\WObj:=wPaper;
    MoveL Offs(pOrigin,158.8,37.5,0.0),vDraw,z1,tPen\WObj:=wPaper;
    MoveL Offs(pOrigin,159.2,37.5,0.0),vDraw,z1,tPen\WObj:=wPaper;
    MoveL Offs(pOrigin,159.4,37.7,0.0),vDraw,z1,tPen\WObj:=wPaper;
    MoveL Offs(pOrigin,159.9,37.7,0.0),vDraw,z1,tPen\WObj:=wPaper;
    MoveL Offs(pOrigin,160.1,37.9,0.0),vDraw,z1,tPen\WObj:=wPaper;
    MoveL Offs(pOrigin,160.7,37.9,0.0),vDraw,z1,tPen\WObj:=wPaper;
    MoveL Offs(pOrigin,160.9,38.1,0.0),vDraw,z1,tPen\WObj:=wPaper;
    MoveL Offs(pOrigin,161.5,38.1,0.0),vDraw,z1,tPen\WObj:=wPaper;
    MoveL Offs(pOrigin,161.6,38.2,0.0),vDraw,z1,tPen\WObj:=wPaper;
    MoveL Offs(pOrigin,162.4,38.2,0.0),vDraw,z1,tPen\WObj:=wPaper;
    MoveL Offs(pOrigin,162.6,38.4,0.0),vDraw,z1,tPen\WObj:=wPaper;
    MoveL Offs(pOrigin,163.3,38.4,0.0),vDraw,z1,tPen\WObj:=wPaper;
    MoveL Offs(pOrigin,163.5,38.6,0.0),vDraw,z1,tPen\WObj:=wPaper;
    MoveL Offs(pOrigin,164.3,38.6,0.0),vDraw,z1,tPen\WObj:=wPaper;
    MoveL Offs(pOrigin,164.5,38.8,0.0),vDraw,z1,tPen\WObj:=wPaper;
    MoveL Offs(pOrigin,165.4,38.8,0.0),vDraw,z1,tPen\WObj:=wPaper;
    MoveL Offs(pOrigin,165.6,39.0,0.0),vDraw,z1,tPen\WObj:=wPaper;
    MoveL Offs(pOrigin,166.6,39.0,0.0),vDraw,z1,tPen\WObj:=wPaper;
    MoveL Offs(pOrigin,166.7,39.2,0.0),vDraw,z1,tPen\WObj:=wPaper;
  ENDPROC

  PROC Part82()
    MoveL Offs(pOrigin,167.7,39.2,0.0),vDraw,z1,tPen\WObj:=wPaper;
    MoveL Offs(pOrigin,167.9,39.4,0.0),vDraw,z1,tPen\WObj:=wPaper;
    MoveL Offs(pOrigin,169.0,39.4,0.0),vDraw,z1,tPen\WObj:=wPaper;
    MoveL Offs(pOrigin,169.2,39.6,0.0),vDraw,z1,tPen\WObj:=wPaper;
    MoveL Offs(pOrigin,170.3,39.6,0.0),vDraw,z1,tPen\WObj:=wPaper;
    MoveL Offs(pOrigin,170.5,39.8,0.0),vDraw,z1,tPen\WObj:=wPaper;
    MoveL Offs(pOrigin,171.7,39.8,0.0),vDraw,z1,tPen\WObj:=wPaper;
    MoveL Offs(pOrigin,171.8,39.9,0.0),vDraw,z1,tPen\WObj:=wPaper;
    MoveL Offs(pOrigin,173.2,39.9,0.0),vDraw,z1,tPen\WObj:=wPaper;
    MoveL Offs(pOrigin,173.4,40.1,0.0),vDraw,z1,tPen\WObj:=wPaper;
    MoveL Offs(pOrigin,174.7,40.1,0.0),vDraw,z1,tPen\WObj:=wPaper;
    MoveL Offs(pOrigin,174.9,40.3,0.0),vDraw,z1,tPen\WObj:=wPaper;
    MoveL Offs(pOrigin,176.4,40.3,0.0),vDraw,z1,tPen\WObj:=wPaper;
    MoveL Offs(pOrigin,176.6,40.5,0.0),vDraw,z1,tPen\WObj:=wPaper;
    MoveL Offs(pOrigin,178.5,40.5,0.0),vDraw,z1,tPen\WObj:=wPaper;
    MoveL Offs(pOrigin,178.6,40.7,0.0),vDraw,z1,tPen\WObj:=wPaper;
    MoveL Offs(pOrigin,184.3,40.7,0.0),vDraw,z1,tPen\WObj:=wPaper;
    MoveL Offs(pOrigin,184.5,40.5,0.0),vDraw,z1,tPen\WObj:=wPaper;
    MoveL Offs(pOrigin,185.8,40.5,0.0),vDraw,z1,tPen\WObj:=wPaper;
    MoveL Offs(pOrigin,186.0,40.3,0.0),vDraw,z1,tPen\WObj:=wPaper;
    MoveL Offs(pOrigin,187.0,40.3,0.0),vDraw,z1,tPen\WObj:=wPaper;
    MoveL Offs(pOrigin,187.1,40.1,0.0),vDraw,z1,tPen\WObj:=wPaper;
    MoveL Offs(pOrigin,187.5,40.1,0.0),vDraw,z1,tPen\WObj:=wPaper;
    MoveL Offs(pOrigin,187.7,39.9,0.0),vDraw,z1,tPen\WObj:=wPaper;
    MoveL Offs(pOrigin,188.3,39.9,0.0),vDraw,z1,tPen\WObj:=wPaper;
    MoveL Offs(pOrigin,188.5,39.8,0.0),vDraw,z1,tPen\WObj:=wPaper;
    MoveL Offs(pOrigin,188.8,39.8,0.0),vDraw,z1,tPen\WObj:=wPaper;
    MoveL Offs(pOrigin,189.0,39.6,0.0),vDraw,z1,tPen\WObj:=wPaper;
    MoveL Offs(pOrigin,189.2,39.6,0.0),vDraw,z1,tPen\WObj:=wPaper;
    MoveL Offs(pOrigin,189.4,39.4,0.0),vDraw,z1,tPen\WObj:=wPaper;
    MoveL Offs(pOrigin,189.6,39.4,0.0),vDraw,z1,tPen\WObj:=wPaper;
    MoveL Offs(pOrigin,189.8,39.2,0.0),vDraw,z1,tPen\WObj:=wPaper;
    MoveL Offs(pOrigin,190.0,39.2,0.0),vDraw,z1,tPen\WObj:=wPaper;
    MoveL Offs(pOrigin,190.2,39.0,0.0),vDraw,z1,tPen\WObj:=wPaper;
    MoveL Offs(pOrigin,191.5,38.4,0.0),vDraw,z1,tPen\WObj:=wPaper;
    MoveL Offs(pOrigin,191.9,38.1,0.0),vDraw,z1,tPen\WObj:=wPaper;
    MoveL Offs(pOrigin,192.1,38.1,0.0),vDraw,z1,tPen\WObj:=wPaper;
    MoveL Offs(pOrigin,192.4,37.7,0.0),vDraw,z1,tPen\WObj:=wPaper;
    MoveL Offs(pOrigin,192.6,37.7,0.0),vDraw,z1,tPen\WObj:=wPaper;
    MoveL Offs(pOrigin,193.2,37.1,0.0),vDraw,z1,tPen\WObj:=wPaper;
    MoveL Offs(pOrigin,193.4,37.1,0.0),vDraw,z1,tPen\WObj:=wPaper;
    MoveL Offs(pOrigin,194.1,36.4,0.0),vDraw,z1,tPen\WObj:=wPaper;
    MoveL Offs(pOrigin,194.3,36.4,0.0),vDraw,z1,tPen\WObj:=wPaper;
    MoveL Offs(pOrigin,197.0,33.7,0.0),vDraw,z1,tPen\WObj:=wPaper;
    MoveL Offs(pOrigin,197.0,33.5,0.0),vDraw,z1,tPen\WObj:=wPaper;
    MoveL Offs(pOrigin,197.7,32.8,0.0),vDraw,z1,tPen\WObj:=wPaper;
    MoveL Offs(pOrigin,197.7,32.6,0.0),vDraw,z1,tPen\WObj:=wPaper;
    MoveL Offs(pOrigin,198.9,31.1,0.0),vDraw,z1,tPen\WObj:=wPaper;
    MoveL Offs(pOrigin,199.0,30.5,0.0),vDraw,z1,tPen\WObj:=wPaper;
    MoveL Offs(pOrigin,199.4,30.1,0.0),vDraw,z1,tPen\WObj:=wPaper;
    MoveL Offs(pOrigin,199.4,29.9,0.0),vDraw,z1,tPen\WObj:=wPaper;
    MoveL Offs(pOrigin,200.0,29.0,0.0),vDraw,z1,tPen\WObj:=wPaper;
    MoveL Offs(pOrigin,200.0,28.6,0.0),vDraw,z1,tPen\WObj:=wPaper;
    MoveL Offs(pOrigin,200.2,28.4,0.0),vDraw,z1,tPen\WObj:=wPaper;
    MoveL Offs(pOrigin,200.2,28.2,0.0),vDraw,z1,tPen\WObj:=wPaper;
    MoveL Offs(pOrigin,200.4,28.0,0.0),vDraw,z1,tPen\WObj:=wPaper;
    MoveL Offs(pOrigin,200.4,27.7,0.0),vDraw,z1,tPen\WObj:=wPaper;
    MoveL Offs(pOrigin,200.6,27.5,0.0),vDraw,z1,tPen\WObj:=wPaper;
    MoveL Offs(pOrigin,200.6,26.9,0.0),vDraw,z1,tPen\WObj:=wPaper;
    MoveL Offs(pOrigin,200.7,26.7,0.0),vDraw,z1,tPen\WObj:=wPaper;
    MoveL Offs(pOrigin,200.7,26.2,0.0),vDraw,z1,tPen\WObj:=wPaper;
    MoveL Offs(pOrigin,200.9,26.0,0.0),vDraw,z1,tPen\WObj:=wPaper;
    MoveL Offs(pOrigin,200.9,25.4,0.0),vDraw,z1,tPen\WObj:=wPaper;
    MoveL Offs(pOrigin,201.1,25.4,0.0),vDraw,z1,tPen\WObj:=wPaper;
    MoveL Offs(pOrigin,201.1,25.6,0.0),vDraw,z1,tPen\WObj:=wPaper;
    MoveL Offs(pOrigin,200.9,25.8,0.0),vDraw,z1,tPen\WObj:=wPaper;
    MoveL Offs(pOrigin,200.9,26.9,0.0),vDraw,z1,tPen\WObj:=wPaper;
    MoveL Offs(pOrigin,200.7,27.1,0.0),vDraw,z1,tPen\WObj:=wPaper;
    MoveL Offs(pOrigin,200.7,27.5,0.0),vDraw,z1,tPen\WObj:=wPaper;
    MoveL Offs(pOrigin,200.6,27.7,0.0),vDraw,z1,tPen\WObj:=wPaper;
    MoveL Offs(pOrigin,200.4,28.6,0.0),vDraw,z1,tPen\WObj:=wPaper;
    MoveL Offs(pOrigin,200.0,29.2,0.0),vDraw,z1,tPen\WObj:=wPaper;
    MoveL Offs(pOrigin,200.0,29.6,0.0),vDraw,z1,tPen\WObj:=wPaper;
    MoveL Offs(pOrigin,199.8,29.7,0.0),vDraw,z1,tPen\WObj:=wPaper;
    MoveL Offs(pOrigin,199.4,30.7,0.0),vDraw,z1,tPen\WObj:=wPaper;
    MoveL Offs(pOrigin,199.0,31.1,0.0),vDraw,z1,tPen\WObj:=wPaper;
    MoveL Offs(pOrigin,198.9,31.6,0.0),vDraw,z1,tPen\WObj:=wPaper;
    MoveL Offs(pOrigin,198.5,32.0,0.0),vDraw,z1,tPen\WObj:=wPaper;
    MoveL Offs(pOrigin,198.5,32.2,0.0),vDraw,z1,tPen\WObj:=wPaper;
    MoveL Offs(pOrigin,198.1,32.6,0.0),vDraw,z1,tPen\WObj:=wPaper;
    MoveL Offs(pOrigin,198.1,32.8,0.0),vDraw,z1,tPen\WObj:=wPaper;
    MoveL Offs(pOrigin,197.3,33.5,0.0),vDraw,z1,tPen\WObj:=wPaper;
    MoveL Offs(pOrigin,197.3,33.7,0.0),vDraw,z1,tPen\WObj:=wPaper;
    MoveL Offs(pOrigin,196.0,35.0,0.0),vDraw,z1,tPen\WObj:=wPaper;
    MoveL Offs(pOrigin,196.0,35.2,0.0),vDraw,z1,tPen\WObj:=wPaper;
    MoveL Offs(pOrigin,195.6,35.6,0.0),vDraw,z1,tPen\WObj:=wPaper;
    MoveL Offs(pOrigin,195.5,35.6,0.0),vDraw,z1,tPen\WObj:=wPaper;
    MoveL Offs(pOrigin,194.1,36.9,0.0),vDraw,z1,tPen\WObj:=wPaper;
    MoveL Offs(pOrigin,193.9,36.9,0.0),vDraw,z1,tPen\WObj:=wPaper;
    MoveL Offs(pOrigin,193.4,37.5,0.0),vDraw,z1,tPen\WObj:=wPaper;
    MoveL Offs(pOrigin,193.2,37.5,0.0),vDraw,z1,tPen\WObj:=wPaper;
    MoveL Offs(pOrigin,192.8,37.9,0.0),vDraw,z1,tPen\WObj:=wPaper;
    MoveL Offs(pOrigin,192.6,37.9,0.0),vDraw,z1,tPen\WObj:=wPaper;
    MoveL Offs(pOrigin,192.1,38.4,0.0),vDraw,z1,tPen\WObj:=wPaper;
    MoveL Offs(pOrigin,191.9,38.4,0.0),vDraw,z1,tPen\WObj:=wPaper;
    MoveL Offs(pOrigin,189.8,39.6,0.0),vDraw,z1,tPen\WObj:=wPaper;
    MoveL Offs(pOrigin,189.4,39.6,0.0),vDraw,z1,tPen\WObj:=wPaper;
    MoveL Offs(pOrigin,188.8,39.9,0.0),vDraw,z1,tPen\WObj:=wPaper;
    MoveL Offs(pOrigin,188.5,39.9,0.0),vDraw,z1,tPen\WObj:=wPaper;
    MoveL Offs(pOrigin,188.3,40.1,0.0),vDraw,z1,tPen\WObj:=wPaper;
    MoveL Offs(pOrigin,187.9,40.1,0.0),vDraw,z1,tPen\WObj:=wPaper;
    MoveL Offs(pOrigin,187.7,40.3,0.0),vDraw,z1,tPen\WObj:=wPaper;
    MoveL Offs(pOrigin,187.3,40.3,0.0),vDraw,z1,tPen\WObj:=wPaper;
    MoveL Offs(pOrigin,187.1,40.5,0.0),vDraw,z1,tPen\WObj:=wPaper;
    MoveL Offs(pOrigin,186.4,40.5,0.0),vDraw,z1,tPen\WObj:=wPaper;
    MoveL Offs(pOrigin,186.2,40.7,0.0),vDraw,z1,tPen\WObj:=wPaper;
    MoveL Offs(pOrigin,185.6,40.7,0.0),vDraw,z1,tPen\WObj:=wPaper;
    MoveL Offs(pOrigin,185.4,40.9,0.0),vDraw,z1,tPen\WObj:=wPaper;
    MoveL Offs(pOrigin,184.5,40.9,0.0),vDraw,z1,tPen\WObj:=wPaper;
    MoveL Offs(pOrigin,184.3,41.1,0.0),vDraw,z1,tPen\WObj:=wPaper;
    MoveL Offs(pOrigin,182.6,41.1,0.0),vDraw,z1,tPen\WObj:=wPaper;
    MoveL Offs(pOrigin,182.4,41.3,0.0),vDraw,z1,tPen\WObj:=wPaper;
    MoveL Offs(pOrigin,181.9,41.3,0.0),vDraw,z1,tPen\WObj:=wPaper;
    MoveL Offs(pOrigin,181.7,41.5,0.0),vDraw,z1,tPen\WObj:=wPaper;
    MoveL Offs(pOrigin,182.2,42.0,0.0),vDraw,z1,tPen\WObj:=wPaper;
    MoveL Offs(pOrigin,182.4,42.0,0.0),vDraw,z1,tPen\WObj:=wPaper;
    MoveL Offs(pOrigin,183.0,42.4,0.0),vDraw,z1,tPen\WObj:=wPaper;
    MoveL Offs(pOrigin,183.6,42.4,0.0),vDraw,z1,tPen\WObj:=wPaper;
    MoveL Offs(pOrigin,183.9,43.0,0.0),vDraw,z1,tPen\WObj:=wPaper;
    MoveL Offs(pOrigin,184.1,43.0,0.0),vDraw,z1,tPen\WObj:=wPaper;
  ENDPROC

  PROC Part83()
    MoveL Offs(pOrigin,185.8,43.9,0.0),vDraw,z1,tPen\WObj:=wPaper;
    MoveL Offs(pOrigin,186.2,43.9,0.0),vDraw,z1,tPen\WObj:=wPaper;
    MoveL Offs(pOrigin,186.4,44.1,0.0),vDraw,z1,tPen\WObj:=wPaper;
    MoveL Offs(pOrigin,186.8,44.1,0.0),vDraw,z1,tPen\WObj:=wPaper;
    MoveL Offs(pOrigin,187.0,44.3,0.0),vDraw,z1,tPen\WObj:=wPaper;
    MoveL Offs(pOrigin,187.5,44.3,0.0),vDraw,z1,tPen\WObj:=wPaper;
    MoveL Offs(pOrigin,187.7,44.5,0.0),vDraw,z1,tPen\WObj:=wPaper;
    MoveL Offs(pOrigin,188.8,44.5,0.0),vDraw,z1,tPen\WObj:=wPaper;
    MoveL Offs(pOrigin,189.0,44.7,0.0),vDraw,z1,tPen\WObj:=wPaper;
    MoveL Offs(pOrigin,189.8,44.7,0.0),vDraw,z1,tPen\WObj:=wPaper;
    MoveL Offs(pOrigin,190.0,44.5,0.0),vDraw,z1,tPen\WObj:=wPaper;
    MoveL Offs(pOrigin,191.7,44.5,0.0),vDraw,z1,tPen\WObj:=wPaper;
    MoveL Offs(pOrigin,191.9,44.3,0.0),vDraw,z1,tPen\WObj:=wPaper;
    MoveL Offs(pOrigin,192.6,44.3,0.0),vDraw,z1,tPen\WObj:=wPaper;
    MoveL Offs(pOrigin,192.8,44.1,0.0),vDraw,z1,tPen\WObj:=wPaper;
    MoveL Offs(pOrigin,193.4,44.1,0.0),vDraw,z1,tPen\WObj:=wPaper;
    MoveL Offs(pOrigin,193.6,43.9,0.0),vDraw,z1,tPen\WObj:=wPaper;
    MoveL Offs(pOrigin,193.9,43.9,0.0),vDraw,z1,tPen\WObj:=wPaper;
    MoveL Offs(pOrigin,194.1,43.7,0.0),vDraw,z1,tPen\WObj:=wPaper;
    MoveL Offs(pOrigin,194.5,43.7,0.0),vDraw,z1,tPen\WObj:=wPaper;
    MoveL Offs(pOrigin,194.7,43.5,0.0),vDraw,z1,tPen\WObj:=wPaper;
    MoveL Offs(pOrigin,195.6,43.3,0.0),vDraw,z1,tPen\WObj:=wPaper;
    MoveL Offs(pOrigin,196.2,43.0,0.0),vDraw,z1,tPen\WObj:=wPaper;
    MoveL Offs(pOrigin,196.6,43.0,0.0),vDraw,z1,tPen\WObj:=wPaper;
    MoveL Offs(pOrigin,196.8,42.8,0.0),vDraw,z1,tPen\WObj:=wPaper;
    MoveL Offs(pOrigin,197.0,42.8,0.0),vDraw,z1,tPen\WObj:=wPaper;
    MoveL Offs(pOrigin,197.2,42.6,0.0),vDraw,z1,tPen\WObj:=wPaper;
    MoveL Offs(pOrigin,197.3,42.6,0.0),vDraw,z1,tPen\WObj:=wPaper;
    MoveL Offs(pOrigin,197.5,42.4,0.0),vDraw,z1,tPen\WObj:=wPaper;
    MoveL Offs(pOrigin,197.7,42.4,0.0),vDraw,z1,tPen\WObj:=wPaper;
    MoveL Offs(pOrigin,197.9,42.2,0.0),vDraw,z1,tPen\WObj:=wPaper;
    MoveL Offs(pOrigin,198.1,42.2,0.0),vDraw,z1,tPen\WObj:=wPaper;
    MoveL Offs(pOrigin,198.3,42.0,0.0),vDraw,z1,tPen\WObj:=wPaper;
    MoveL Offs(pOrigin,199.6,41.5,0.0),vDraw,z1,tPen\WObj:=wPaper;
    MoveL Offs(pOrigin,200.0,41.1,0.0),vDraw,z1,tPen\WObj:=wPaper;
    MoveL Offs(pOrigin,200.6,40.9,0.0),vDraw,z1,tPen\WObj:=wPaper;
    MoveL Offs(pOrigin,200.9,40.5,0.0),vDraw,z1,tPen\WObj:=wPaper;
    MoveL Offs(pOrigin,201.1,40.5,0.0),vDraw,z1,tPen\WObj:=wPaper;
    MoveL Offs(pOrigin,201.5,40.1,0.0),vDraw,z1,tPen\WObj:=wPaper;
    MoveL Offs(pOrigin,201.7,40.1,0.0),vDraw,z1,tPen\WObj:=wPaper;
    MoveL Offs(pOrigin,202.1,39.8,0.0),vDraw,z1,tPen\WObj:=wPaper;
    MoveL Offs(pOrigin,202.3,39.8,0.0),vDraw,z1,tPen\WObj:=wPaper;
    MoveL Offs(pOrigin,203.0,39.0,0.0),vDraw,z1,tPen\WObj:=wPaper;
    MoveL Offs(pOrigin,203.2,39.0,0.0),vDraw,z1,tPen\WObj:=wPaper;
    MoveL Offs(pOrigin,204.5,37.7,0.0),vDraw,z1,tPen\WObj:=wPaper;
    MoveL Offs(pOrigin,204.7,37.7,0.0),vDraw,z1,tPen\WObj:=wPaper;
    MoveL Offs(pOrigin,206.4,35.6,0.0),vDraw,z1,tPen\WObj:=wPaper;
    MoveL Offs(pOrigin,206.4,35.4,0.0),vDraw,z1,tPen\WObj:=wPaper;
    MoveL Offs(pOrigin,207.0,34.5,0.0),vDraw,z1,tPen\WObj:=wPaper;
    MoveL Offs(pOrigin,207.0,33.9,0.0),vDraw,z1,tPen\WObj:=wPaper;
    MoveL Offs(pOrigin,207.2,33.7,0.0),vDraw,z1,tPen\WObj:=wPaper;
    MoveL Offs(pOrigin,207.2,32.8,0.0),vDraw,z1,tPen\WObj:=wPaper;
    MoveL Offs(pOrigin,207.4,32.6,0.0),vDraw,z1,tPen\WObj:=wPaper;
    MoveL Offs(pOrigin,207.4,29.6,0.0),vDraw,z1,tPen\WObj:=wPaper;
    MoveL Offs(pOrigin,207.2,29.4,0.0),vDraw,z1,tPen\WObj:=wPaper;
    MoveL Offs(pOrigin,207.2,28.6,0.0),vDraw,z1,tPen\WObj:=wPaper;
    MoveL Offs(pOrigin,207.0,28.4,0.0),vDraw,z1,tPen\WObj:=wPaper;
    MoveL Offs(pOrigin,207.0,27.9,0.0),vDraw,z1,tPen\WObj:=wPaper;
    MoveL Offs(pOrigin,206.8,27.7,0.0),vDraw,z1,tPen\WObj:=wPaper;
    MoveL Offs(pOrigin,206.6,26.7,0.0),vDraw,z1,tPen\WObj:=wPaper;
    MoveL Offs(pOrigin,206.4,26.5,0.0),vDraw,z1,tPen\WObj:=wPaper;
    MoveL Offs(pOrigin,206.0,25.6,0.0),vDraw,z1,tPen\WObj:=wPaper;
    MoveL Offs(pOrigin,205.7,25.2,0.0),vDraw,z1,tPen\WObj:=wPaper;
    MoveL Offs(pOrigin,205.7,25.0,0.0),vDraw,z1,tPen\WObj:=wPaper;
    MoveL Offs(pOrigin,204.5,23.9,0.0),vDraw,z1,tPen\WObj:=wPaper;
    MoveL Offs(pOrigin,204.3,24.1,0.0),vDraw,z1,tPen\WObj:=wPaper;
    MoveL Offs(pOrigin,204.3,24.5,0.0),vDraw,z1,tPen\WObj:=wPaper;
    MoveL Offs(pOrigin,204.5,24.6,0.0),vDraw,z1,tPen\WObj:=wPaper;
    MoveL Offs(pOrigin,204.5,25.0,0.0),vDraw,z1,tPen\WObj:=wPaper;
    MoveL Offs(pOrigin,204.7,25.2,0.0),vDraw,z1,tPen\WObj:=wPaper;
    MoveL Offs(pOrigin,204.7,25.6,0.0),vDraw,z1,tPen\WObj:=wPaper;
    MoveL Offs(pOrigin,204.9,25.8,0.0),vDraw,z1,tPen\WObj:=wPaper;
    MoveL Offs(pOrigin,204.9,26.7,0.0),vDraw,z1,tPen\WObj:=wPaper;
    MoveL Offs(pOrigin,205.1,26.9,0.0),vDraw,z1,tPen\WObj:=wPaper;
    MoveL Offs(pOrigin,205.1,29.9,0.0),vDraw,z1,tPen\WObj:=wPaper;
    MoveL Offs(pOrigin,204.9,30.1,0.0),vDraw,z1,tPen\WObj:=wPaper;
    MoveL Offs(pOrigin,204.9,31.1,0.0),vDraw,z1,tPen\WObj:=wPaper;
    MoveL Offs(pOrigin,204.7,31.3,0.0),vDraw,z1,tPen\WObj:=wPaper;
    MoveL Offs(pOrigin,204.7,31.8,0.0),vDraw,z1,tPen\WObj:=wPaper;
    MoveL Offs(pOrigin,204.5,32.0,0.0),vDraw,z1,tPen\WObj:=wPaper;
    MoveL Offs(pOrigin,204.5,32.6,0.0),vDraw,z1,tPen\WObj:=wPaper;
    MoveL Offs(pOrigin,204.3,32.8,0.0),vDraw,z1,tPen\WObj:=wPaper;
    MoveL Offs(pOrigin,204.3,33.1,0.0),vDraw,z1,tPen\WObj:=wPaper;
    MoveL Offs(pOrigin,203.6,34.5,0.0),vDraw,z1,tPen\WObj:=wPaper;
    MoveL Offs(pOrigin,203.6,34.8,0.0),vDraw,z1,tPen\WObj:=wPaper;
    MoveL Offs(pOrigin,203.4,35.0,0.0),vDraw,z1,tPen\WObj:=wPaper;
    MoveL Offs(pOrigin,203.0,36.0,0.0),vDraw,z1,tPen\WObj:=wPaper;
    MoveL Offs(pOrigin,202.6,36.4,0.0),vDraw,z1,tPen\WObj:=wPaper;
    MoveL Offs(pOrigin,202.4,36.9,0.0),vDraw,z1,tPen\WObj:=wPaper;
    MoveL Offs(pOrigin,202.1,37.3,0.0),vDraw,z1,tPen\WObj:=wPaper;
    MoveL Offs(pOrigin,202.1,37.5,0.0),vDraw,z1,tPen\WObj:=wPaper;
    MoveL Offs(pOrigin,201.9,37.5,0.0),vDraw,z1,tPen\WObj:=wPaper;
    MoveL Offs(pOrigin,202.1,37.3,0.0),vDraw,z1,tPen\WObj:=wPaper;
    MoveL Offs(pOrigin,202.1,37.1,0.0),vDraw,z1,tPen\WObj:=wPaper;
    MoveL Offs(pOrigin,202.3,36.9,0.0),vDraw,z1,tPen\WObj:=wPaper;
    MoveL Offs(pOrigin,202.3,36.7,0.0),vDraw,z1,tPen\WObj:=wPaper;
    MoveL Offs(pOrigin,202.4,36.5,0.0),vDraw,z1,tPen\WObj:=wPaper;
    MoveL Offs(pOrigin,202.4,36.4,0.0),vDraw,z1,tPen\WObj:=wPaper;
    MoveL Offs(pOrigin,203.6,34.3,0.0),vDraw,z1,tPen\WObj:=wPaper;
    MoveL Offs(pOrigin,203.6,33.9,0.0),vDraw,z1,tPen\WObj:=wPaper;
    MoveL Offs(pOrigin,203.8,33.7,0.0),vDraw,z1,tPen\WObj:=wPaper;
    MoveL Offs(pOrigin,203.8,33.3,0.0),vDraw,z1,tPen\WObj:=wPaper;
    MoveL Offs(pOrigin,204.0,33.1,0.0),vDraw,z1,tPen\WObj:=wPaper;
    MoveL Offs(pOrigin,204.0,32.8,0.0),vDraw,z1,tPen\WObj:=wPaper;
    MoveL Offs(pOrigin,204.1,32.6,0.0),vDraw,z1,tPen\WObj:=wPaper;
    MoveL Offs(pOrigin,204.1,32.2,0.0),vDraw,z1,tPen\WObj:=wPaper;
    MoveL Offs(pOrigin,204.3,32.0,0.0),vDraw,z1,tPen\WObj:=wPaper;
    MoveL Offs(pOrigin,204.3,31.3,0.0),vDraw,z1,tPen\WObj:=wPaper;
    MoveL Offs(pOrigin,204.5,31.1,0.0),vDraw,z1,tPen\WObj:=wPaper;
    MoveL Offs(pOrigin,204.5,30.1,0.0),vDraw,z1,tPen\WObj:=wPaper;
    MoveL Offs(pOrigin,204.7,29.9,0.0),vDraw,z1,tPen\WObj:=wPaper;
    MoveL Offs(pOrigin,204.7,26.9,0.0),vDraw,z1,tPen\WObj:=wPaper;
    MoveL Offs(pOrigin,204.5,26.7,0.0),vDraw,z1,tPen\WObj:=wPaper;
    MoveL Offs(pOrigin,204.5,25.8,0.0),vDraw,z1,tPen\WObj:=wPaper;
    MoveL Offs(pOrigin,204.3,25.6,0.0),vDraw,z1,tPen\WObj:=wPaper;
    MoveL Offs(pOrigin,204.3,25.2,0.0),vDraw,z1,tPen\WObj:=wPaper;
    MoveL Offs(pOrigin,204.1,25.0,0.0),vDraw,z1,tPen\WObj:=wPaper;
    MoveL Offs(pOrigin,204.0,24.1,0.0),vDraw,z1,tPen\WObj:=wPaper;
    MoveL Offs(pOrigin,203.8,23.9,0.0),vDraw,z1,tPen\WObj:=wPaper;
    MoveL Offs(pOrigin,203.6,23.3,0.0),vDraw,z1,tPen\WObj:=wPaper;
  ENDPROC

  PROC Part84()
    MoveL Offs(pOrigin,203.0,22.8,0.0),vDraw,z1,tPen\WObj:=wPaper;
    MoveL Offs(pOrigin,202.8,22.8,0.0),vDraw,z1,tPen\WObj:=wPaper;
    MoveL Offs(pOrigin,202.6,22.6,0.0),vDraw,z1,tPen\WObj:=wPaper;
    MoveL Offs(pOrigin,202.3,22.6,0.0),vDraw,z1,tPen\WObj:=wPaper;
    MoveL Offs(pOrigin,201.7,22.2,0.0),vDraw,z1,tPen\WObj:=wPaper;
    MoveL Offs(pOrigin,201.3,22.2,0.0),vDraw,z1,tPen\WObj:=wPaper;
    MoveL Offs(pOrigin,201.1,22.0,0.0),vDraw,z1,tPen\WObj:=wPaper;
    MoveL Offs(pOrigin,200.7,22.0,0.0),vDraw,z1,tPen\WObj:=wPaper;
    MoveL Offs(pOrigin,200.6,21.8,0.0),vDraw,z1,tPen\WObj:=wPaper;
    MoveL Offs(pOrigin,199.6,21.6,0.0),vDraw,z1,tPen\WObj:=wPaper;
    MoveL Offs(pOrigin,199.4,21.4,0.0),vDraw,z1,tPen\WObj:=wPaper;
    MoveL Offs(pOrigin,198.9,21.4,0.0),vDraw,z1,tPen\WObj:=wPaper;
    MoveL Offs(pOrigin,198.7,21.2,0.0),vDraw,z1,tPen\WObj:=wPaper;
    MoveL Offs(pOrigin,198.3,21.2,0.0),vDraw,z1,tPen\WObj:=wPaper;
    MoveL Offs(pOrigin,198.1,21.1,0.0),vDraw,z1,tPen\WObj:=wPaper;
    MoveL Offs(pOrigin,197.3,21.1,0.0),vDraw,z1,tPen\WObj:=wPaper;
    MoveL Offs(pOrigin,197.2,20.9,0.0),vDraw,z1,tPen\WObj:=wPaper;
    MoveL Offs(pOrigin,196.6,20.9,0.0),vDraw,z1,tPen\WObj:=wPaper;
    MoveL Offs(pOrigin,196.4,20.7,0.0),vDraw,z1,tPen\WObj:=wPaper;
    MoveL Offs(pOrigin,195.6,20.7,0.0),vDraw,z1,tPen\WObj:=wPaper;
    MoveL Offs(pOrigin,195.5,20.5,0.0),vDraw,z1,tPen\WObj:=wPaper;
    MoveL Offs(pOrigin,194.5,20.5,0.0),vDraw,z1,tPen\WObj:=wPaper;
    MoveL Offs(pOrigin,194.3,20.3,0.0),vDraw,z1,tPen\WObj:=wPaper;
    MoveL Offs(pOrigin,193.6,20.3,0.0),vDraw,z1,tPen\WObj:=wPaper;
    MoveL Offs(pOrigin,193.4,20.1,0.0),vDraw,z1,tPen\WObj:=wPaper;
    MoveL Offs(pOrigin,192.4,20.1,0.0),vDraw,z1,tPen\WObj:=wPaper;
    MoveL Offs(pOrigin,192.2,19.9,0.0),vDraw,z1,tPen\WObj:=wPaper;
    MoveL Offs(pOrigin,191.1,19.9,0.0),vDraw,z1,tPen\WObj:=wPaper;
    MoveL Offs(pOrigin,190.9,19.7,0.0),vDraw,z1,tPen\WObj:=wPaper;
    MoveL Offs(pOrigin,189.8,19.7,0.0),vDraw,z1,tPen\WObj:=wPaper;
    MoveL Offs(pOrigin,189.6,19.5,0.0),vDraw,z1,tPen\WObj:=wPaper;
    MoveL Offs(pOrigin,188.5,19.5,0.0),vDraw,z1,tPen\WObj:=wPaper;
    MoveL Offs(pOrigin,188.3,19.4,0.0),vDraw,z1,tPen\WObj:=wPaper;
    MoveL Offs(pOrigin,187.0,19.4,0.0),vDraw,z1,tPen\WObj:=wPaper;
    MoveL Offs(pOrigin,186.8,19.2,0.0),vDraw,z1,tPen\WObj:=wPaper;
    MoveL Offs(pOrigin,185.4,19.2,0.0),vDraw,z1,tPen\WObj:=wPaper;
    MoveL Offs(pOrigin,185.3,19.0,0.0),vDraw,z1,tPen\WObj:=wPaper;
    MoveL Offs(pOrigin,184.3,19.0,0.0),vDraw,z1,tPen\WObj:=wPaper;
    MoveL Offs(pOrigin,184.1,19.2,0.0),vDraw,z1,tPen\WObj:=wPaper;
    MoveL Offs(pOrigin,184.3,19.4,0.0),vDraw,z1,tPen\WObj:=wPaper;
    MoveL Offs(pOrigin,184.5,19.4,0.0),vDraw,z1,tPen\WObj:=wPaper;
    MoveL Offs(pOrigin,184.7,19.5,0.0),vDraw,z1,tPen\WObj:=wPaper;
    MoveL Offs(pOrigin,185.1,19.5,0.0),vDraw,z1,tPen\WObj:=wPaper;
    MoveL Offs(pOrigin,185.6,19.9,0.0),vDraw,z1,tPen\WObj:=wPaper;
    MoveL Offs(pOrigin,186.0,19.9,0.0),vDraw,z1,tPen\WObj:=wPaper;
    MoveL Offs(pOrigin,186.2,20.1,0.0),vDraw,z1,tPen\WObj:=wPaper;
    MoveL Offs(pOrigin,186.6,20.1,0.0),vDraw,z1,tPen\WObj:=wPaper;
    MoveL Offs(pOrigin,186.8,20.3,0.0),vDraw,z1,tPen\WObj:=wPaper;
    MoveL Offs(pOrigin,187.1,20.3,0.0),vDraw,z1,tPen\WObj:=wPaper;
    MoveL Offs(pOrigin,187.3,20.5,0.0),vDraw,z1,tPen\WObj:=wPaper;
    MoveL Offs(pOrigin,187.7,20.5,0.0),vDraw,z1,tPen\WObj:=wPaper;
    MoveL Offs(pOrigin,187.9,20.7,0.0),vDraw,z1,tPen\WObj:=wPaper;
    MoveL Offs(pOrigin,188.3,20.7,0.0),vDraw,z1,tPen\WObj:=wPaper;
    MoveL Offs(pOrigin,188.5,20.9,0.0),vDraw,z1,tPen\WObj:=wPaper;
    MoveL Offs(pOrigin,188.8,20.9,0.0),vDraw,z1,tPen\WObj:=wPaper;
    MoveL Offs(pOrigin,189.0,21.1,0.0),vDraw,z1,tPen\WObj:=wPaper;
    MoveL Offs(pOrigin,189.4,21.1,0.0),vDraw,z1,tPen\WObj:=wPaper;
    MoveL Offs(pOrigin,189.6,21.2,0.0),vDraw,z1,tPen\WObj:=wPaper;
    MoveL Offs(pOrigin,190.0,21.2,0.0),vDraw,z1,tPen\WObj:=wPaper;
    MoveL Offs(pOrigin,190.2,21.4,0.0),vDraw,z1,tPen\WObj:=wPaper;
    MoveL Offs(pOrigin,191.1,21.6,0.0),vDraw,z1,tPen\WObj:=wPaper;
    MoveL Offs(pOrigin,190.0,21.6,0.0),vDraw,z1,tPen\WObj:=wPaper;
    MoveL Offs(pOrigin,189.8,21.4,0.0),vDraw,z1,tPen\WObj:=wPaper;
    MoveL Offs(pOrigin,189.0,21.4,0.0),vDraw,z1,tPen\WObj:=wPaper;
    MoveL Offs(pOrigin,188.8,21.2,0.0),vDraw,z1,tPen\WObj:=wPaper;
    MoveL Offs(pOrigin,188.3,21.2,0.0),vDraw,z1,tPen\WObj:=wPaper;
    MoveL Offs(pOrigin,188.1,21.1,0.0),vDraw,z1,tPen\WObj:=wPaper;
    MoveL Offs(pOrigin,187.5,21.1,0.0),vDraw,z1,tPen\WObj:=wPaper;
    MoveL Offs(pOrigin,187.3,20.9,0.0),vDraw,z1,tPen\WObj:=wPaper;
    MoveL Offs(pOrigin,187.0,20.9,0.0),vDraw,z1,tPen\WObj:=wPaper;
    MoveL Offs(pOrigin,186.8,20.7,0.0),vDraw,z1,tPen\WObj:=wPaper;
    MoveL Offs(pOrigin,186.4,20.7,0.0),vDraw,z1,tPen\WObj:=wPaper;
    MoveL Offs(pOrigin,186.2,20.5,0.0),vDraw,z1,tPen\WObj:=wPaper;
    MoveL Offs(pOrigin,185.6,20.5,0.0),vDraw,z1,tPen\WObj:=wPaper;
    MoveL Offs(pOrigin,185.4,20.3,0.0),vDraw,z1,tPen\WObj:=wPaper;
    MoveL Offs(pOrigin,185.1,20.3,0.0),vDraw,z1,tPen\WObj:=wPaper;
    MoveL Offs(pOrigin,184.9,20.1,0.0),vDraw,z1,tPen\WObj:=wPaper;
    MoveL Offs(pOrigin,183.9,19.9,0.0),vDraw,z1,tPen\WObj:=wPaper;
    MoveL Offs(pOrigin,183.4,19.5,0.0),vDraw,z1,tPen\WObj:=wPaper;
    MoveL Offs(pOrigin,182.4,19.4,0.0),vDraw,z1,tPen\WObj:=wPaper;
    MoveL Offs(pOrigin,182.2,19.2,0.0),vDraw,z1,tPen\WObj:=wPaper;
    MoveL Offs(pOrigin,182.0,19.2,0.0),vDraw,z1,tPen\WObj:=wPaper;
    MoveL Offs(pOrigin,181.9,19.0,0.0),vDraw,z1,tPen\WObj:=wPaper;
    MoveL Offs(pOrigin,181.5,19.0,0.0),vDraw,z1,tPen\WObj:=wPaper;
    MoveL Offs(pOrigin,180.2,18.2,0.0),vDraw,z1,tPen\WObj:=wPaper;
    MoveL Offs(pOrigin,179.8,18.2,0.0),vDraw,z1,tPen\WObj:=wPaper;
    MoveL Offs(pOrigin,179.6,18.0,0.0),vDraw,z1,tPen\WObj:=wPaper;
    MoveL Offs(pOrigin,179.4,18.0,0.0),vDraw,z1,tPen\WObj:=wPaper;
    MoveL Offs(pOrigin,179.2,17.8,0.0),vDraw,z1,tPen\WObj:=wPaper;
    MoveL Offs(pOrigin,179.0,17.8,0.0),vDraw,z1,tPen\WObj:=wPaper;
    MoveL Offs(pOrigin,176.9,16.7,0.0),vDraw,z1,tPen\WObj:=wPaper;
    MoveL Offs(pOrigin,176.6,16.7,0.0),vDraw,z1,tPen\WObj:=wPaper;
    MoveL Offs(pOrigin,175.6,16.1,0.0),vDraw,z1,tPen\WObj:=wPaper;
    MoveL Offs(pOrigin,175.2,16.1,0.0),vDraw,z1,tPen\WObj:=wPaper;
    MoveL Offs(pOrigin,174.7,15.8,0.0),vDraw,z1,tPen\WObj:=wPaper;
    MoveL Offs(pOrigin,174.1,15.8,0.0),vDraw,z1,tPen\WObj:=wPaper;
    MoveL Offs(pOrigin,173.9,15.6,0.0),vDraw,z1,tPen\WObj:=wPaper;
    MoveL Offs(pOrigin,173.0,15.4,0.0),vDraw,z1,tPen\WObj:=wPaper;
    MoveL Offs(pOrigin,172.8,15.6,0.0),vDraw,z1,tPen\WObj:=wPaper;
    MoveL Offs(pOrigin,174.3,17.1,0.0),vDraw,z1,tPen\WObj:=wPaper;
    MoveL Offs(pOrigin,174.5,17.7,0.0),vDraw,z1,tPen\WObj:=wPaper;
    MoveL Offs(pOrigin,174.9,18.0,0.0),vDraw,z1,tPen\WObj:=wPaper;
    MoveL Offs(pOrigin,174.9,18.4,0.0),vDraw,z1,tPen\WObj:=wPaper;
    MoveL Offs(pOrigin,175.1,18.6,0.0),vDraw,z1,tPen\WObj:=wPaper;
    MoveL Offs(pOrigin,175.1,19.0,0.0),vDraw,z1,tPen\WObj:=wPaper;
    MoveL Offs(pOrigin,175.2,19.2,0.0),vDraw,z1,tPen\WObj:=wPaper;
    MoveL Offs(pOrigin,175.2,19.5,0.0),vDraw,z1,tPen\WObj:=wPaper;
    MoveL Offs(pOrigin,175.4,19.7,0.0),vDraw,z1,tPen\WObj:=wPaper;
    MoveL Offs(pOrigin,175.4,22.0,0.0),vDraw,z1,tPen\WObj:=wPaper;
    MoveL Offs(pOrigin,175.2,22.2,0.0),vDraw,z1,tPen\WObj:=wPaper;
    MoveL Offs(pOrigin,175.2,22.8,0.0),vDraw,z1,tPen\WObj:=wPaper;
    MoveL Offs(pOrigin,175.1,22.9,0.0),vDraw,z1,tPen\WObj:=wPaper;
    MoveL Offs(pOrigin,175.1,23.3,0.0),vDraw,z1,tPen\WObj:=wPaper;
    MoveL Offs(pOrigin,174.7,23.9,0.0),vDraw,z1,tPen\WObj:=wPaper;
    MoveL Offs(pOrigin,174.7,24.3,0.0),vDraw,z1,tPen\WObj:=wPaper;
    MoveL Offs(pOrigin,174.5,24.5,0.0),vDraw,z1,tPen\WObj:=wPaper;
    MoveL Offs(pOrigin,173.9,25.8,0.0),vDraw,z1,tPen\WObj:=wPaper;
    MoveL Offs(pOrigin,173.5,26.2,0.0),vDraw,z1,tPen\WObj:=wPaper;
    MoveL Offs(pOrigin,173.2,27.1,0.0),vDraw,z1,tPen\WObj:=wPaper;
    MoveL Offs(pOrigin,172.8,27.5,0.0),vDraw,z1,tPen\WObj:=wPaper;
  ENDPROC

